// TwinCAT 3 PLC project Standard
// ProgramVersion: 3.1.4023.0
// libraries:
//   Tc2_MDP, * (Beckhoff Automation GmbH)
//   Tc2_Standard, * (Beckhoff Automation GmbH)
//   Tc2_SUPS, * (Beckhoff Automation GmbH)
//   Tc2_System, * (Beckhoff Automation GmbH)
//   Tc2_Utilities, * (Beckhoff Automation GmbH)
//   Tc3_BA2, * (Beckhoff Automation GmbH)
//   Tc3_BA2_Common, * (Beckhoff Automation GmbH)
//   Tc3_BACnetRev14, * (Beckhoff Automation GmbH)
//   Tc3_Module, * (Beckhoff Automation GmbH)
// project tree:
//   / PlcTask.TcTTO (not stored)
//   POUs/ MAIN.TcPOU (not stored)
//   Templates/DUTs/Enumerations/Building/ E_BA_BuildingMode.TcDUT
//   Templates/DUTs/Enumerations/Plant/AC/ E_BA_AC_OpMod01.TcDUT, E_BA_AC_OpMod02.TcDUT, E_BA_AC_SelSpErc.TcDUT
//   Templates/DUTs/Enumerations/Process/ E_BA_Process.TcDUT
//   Templates/DUTs/Enumerations/System/ E_BA_UPSType.TcDUT
//   Templates/DUTs/Enumerations/Universal/ E_BA_EnergyLvl.TcDUT, E_BA_EnergyLvlA.TcDUT, E_BA_EnergyLvlEx.TcDUT, E_BA_EnergyLvlExA.TcDUT, E_BA_MdltCmd.TcDUT, E_BA_OnOff.TcDUT, E_BA_OnOffA.TcDUT
//   Templates/DUTs/Types/Building/ ST_BA_BuildingAlarms.TcDUT
//   Templates/DUTs/Types/General/ ST_BA_GeneralSettings.TcDUT (not stored)
//   Templates/DUTs/Types/WeatherStation/ ST_BA_WeatherStation.TcDUT
//   Templates/GVLs/ BA2_Param.TcGVL
//   Templates/GVLs/DPAD/EventClasses/ EventClasses.TcGVL
//   Templates/GVLs/DPAD/Labels/1031/ LblAggregates1031.TcGVL, LblControl1031.TcGVL, LblFunctions1031.TcGVL
//   Templates/GVLs/DPAD/Labels/1033/ LblAggregates1033.TcGVL, LblControl1033.TcGVL, LblFunctions1033.TcGVL
//   Templates/GVLs/DPAD/Labels/Base/ LblAggregates.TcGVL (not stored), LblControl.TcGVL (not stored), LblFunctions.TcGVL (not stored)
//   Templates/GVLs/DPAD/Labels/Composition/ LblCmpAC.TcGVL, LblCmpGeneral.TcGVL, LblCmpHeating.TcGVL, LblCmpRoomAutomation.TcGVL, LblUniControl.TcGVL, LblUniFieldDevice.TcGVL
//   Templates/GVLs/DPAD/Texts/1031/ TxtEvent_1031.TcGVL, TxtPlant_1031.TcGVL, TxtTrade_1031.TcGVL
//   Templates/GVLs/DPAD/Texts/ TextPlants.TcGVL (not stored), Texts.TcGVL (not stored), TextTrades.TcGVL (not stored)
//   Templates/GVLs/Site/ Site.TcGVL (not stored)
//   Templates/POUs/Trade/AC/Aggregates/Cooler/Temperature/ FB_BA_AC_ColTSuACtrl.TcPOU, FB_BA_AC_ColT_02.TcPOU
//   Templates/POUs/Trade/AC/Aggregates/ERC/ FB_BA_AC_ErcTSuACtrl.TcPOU
//   Templates/POUs/Trade/AC/Aggregates/ERC/Plate/ FB_BA_AC_ErcPl_02.TcPOU
//   Templates/POUs/Trade/AC/Aggregates/PreHeater/ FB_BA_AC_PreHtr.TcPOU, FB_BA_AC_PreHtrTSuACtrl.TcPOU, FB_BA_AC_TRtCtrl.TcPOU
//   Templates/POUs/Trade/AC/ FB_BA_AC.TcPOU
//   Templates/POUs/Trade/AC/General/ FB_BA_AC_OpMod1St.TcPOU, FB_BA_AC_SumNgtCol.TcPOU
//   Templates/POUs/Trade/AC/Plants/ FB_BA_AHU_1St_PrHtr_ErcPl_Col.TcPOU
//   Templates/POUs/Trade/AC/Setpoint/Temperature/ FB_BA_AC_SpTRm_01.TcPOU, FB_BA_AC_TCasCtrl_01.TcPOU
//   Templates/POUs/Trade/General/Building/ FB_BA_BuildingAlarms.TcPOU, FB_BA_BuildingGlobal.TcPOU (not stored), FB_BA_BuildingMode.TcPOU
//   Templates/POUs/Trade/General/ControlCabinet/ FB_BA_ControlCabinet.TcPOU (not stored), FB_BA_ControlCabinetBasic.TcPOU (not stored)
//   Templates/POUs/Trade/General/EventClasses/ FB_BA_EvtGroups.TcPOU (not stored)
//   Templates/POUs/Trade/General/ FB_BA_General.TcPOU (not stored)
//   Templates/POUs/Trade/General/IFP/ FB_BA_IFP.TcPOU
//   Templates/POUs/Trade/General/IFP/Project/ FB_BA_ProjectEx.TcPOU (not stored)
//   Templates/POUs/Trade/General/Settings/ FB_BA_Settings.TcPOU, FB_BA_WeatherParamter.TcPOU (not stored)
//   Templates/POUs/Trade/HeatingSystem/Distribution/HeatingCircuit/ FB_BA_H_HtgCir01.TcPOU
//   Templates/POUs/Trade/HeatingSystem/ FB_BA_H.TcPOU
//   Templates/POUs/Trade/HeatingSystem/General/ FB_BA_HtgLmt.TcPOU, FB_BA_H_OpMod.TcPOU
//   Templates/POUs/Trade/HeatingSystem/Setpoint/ FB_BA_H_HtgCir_Sp.TcPOU
//   Templates/POUs/Trade/OutdoorDevices/ FB_BA_OD.TcPOU (not stored)
//   Templates/POUs/Universal/Aggregat/Analog/ FB_BA_ActuatorAnalog.TcPOU
//   Templates/POUs/Universal/Aggregat/Binary/ FB_BA_ActuatorCmd.TcPOU (not stored)
//   Templates/POUs/Universal/Control/AntiBlocking/ FB_BA_AntiBlocking.TcPOU
//   Templates/POUs/Universal/Control/EventClasses/ FB_BA_EvtCategory_SimpStand.TcPOU (not stored), FB_BA_EvtCategory_SimpStandExt.TcPOU (not stored)
//   Templates/POUs/Universal/Control/Hysteresis/ FB_BA_Hys_21.TcPOU
//   Templates/POUs/Universal/Control/Monitoring/ FB_BA_FdbAnalog.TcPOU, FB_BA_FdbBinary.TcPOU
//   Templates/POUs/Universal/Control/PID/ FB_BA_PID.TcPOU, FB_BA_PID_Sp.TcPOU
//   Templates/POUs/Universal/Control/Ramp/ FB_BA_RampLimitIncrease.TcPOU
//   Templates/POUs/Universal/Control/Scale/ FB_BA_Scale_02.TcPOU, FB_BA_Scale_04.TcPOU
//   Templates/POUs/Universal/Control/TimeDelay/ FB_BA_DlyOff.TcPOU, FB_BA_DlyOn.TcPOU
//   Templates/POUs/Universal/Control/Trend/ FB_BA_TrendLogging.TcPOU
//   Templates/POUs/Universal/Damper/2P/ FB_BA_Dmp2P.TcPOU
//   Templates/POUs/Universal/Motor/1st/ FB_BA_Mot1st.TcPOU
//   Templates/POUs/Universal/Motor/Control/ FB_BA_MotCtlExt.TcPOU
//   Templates/POUs/Universal/Pump/1st/ FB_BA_Pu1st.TcPOU
//   Templates/POUs/Universal/Sensor/ FB_BA_CombinationBI_BV.TcPOU (not stored), FB_BA_SensorAnalog_IO.TcPOU, FB_BA_SensorBinary_IO.TcPOU
//   Templates/POUs/Universal/Valve/ FB_BA_Vlv.TcPOU

// ---- Templates/DUTs/Enumerations/Building/E_BA_BuildingMode.TcDUT
{region '#Template'}
	{attribute 'Version' := '1.0.0.0'}
	{attribute 'Tags' := '"LCID": "1031", "Text": "DUT, Building, RA, OpMod, Mode"'}
	{attribute 'Tags' := '"LCID": "1033", "Text": "DUT, Building, RA, OpMod, Mode"'}
	{attribute 'Description' := '"LCID": "1031", "Text": "Gebäude-Betriebsart"'}
	{attribute 'Description' := '"LCID": "1033", "Text": "Building-operation-mode"'}
{endregion}

{attribute qualified_only}
TYPE E_BA_BuildingMode :
(
	eDefault		:= 1,
	eNightWatch		:= 2,
	eCleaning		:= 3
	
) UDINT;
END_TYPE

// ---- Templates/DUTs/Enumerations/Plant/AC/E_BA_AC_OpMod01.TcDUT
{region '#Template'}
	{attribute 'Version' := '1.0.0.0'}
	{attribute 'Tags' := '"LCID": "1031", "Text": "DUT, Plant, AC, OpMod"'}
	{attribute 'Tags' := '"LCID": "1033", "Text": "DUT, Plant, AC, OpMod"'}
	{attribute 'Description' := '"LCID": "1031", "Text": "Betriebsart Klimaanlage"'}
	{attribute 'Description' := '"LCID": "1033", "Text": "Operation Mode Air Conditioning"'}
{endregion}

{attribute qualified_only}
TYPE E_BA_AC_OpMod01 :
(
    Invalid							:= 0,
    eOff							:= 1,	// Aus							// Off
	eOn								:= 2,	// Ein							// On
    eEmergency						:= 3,	// Notfall						// Emergency
    eFrost							:= 4,	// Frost						// Frost
    eSmokeExtractionProgramm		:= 5,	// Entrauchung Programm			// Smoke extraction programm
    eSmokeExtractionSupplyAir		:= 6,	// Entrauchung Zuluft			// Smoke extraction supply air
    eSmokeExtractionExhaustAir		:= 7,	// Entrauchung Fortluft			// Smoke extraction exhaust air
    eFire							:= 8,	// Feuer						// Fire
    eNightCooling					:= 9,	// Nachtkühlung					// Night cooling
    eCoolDownProtection				:= 10,	// Stützbetrieb,Auskühlschutz	// Cool down protection
    eOverHeatingProtection			:= 11,	// Überhitzungsschutz			// Over heating protection
    eAlarm							:= 12,	// Störung						// Alarm
    eForcedVentilation				:= 13,	// Zwangsbelüftung				// Forced ventilation
    eCentralSwitchOff				:= 14	// Zentralabschaltung			// Central switch-off
) UDINT;
END_TYPE

// ---- Templates/DUTs/Enumerations/Plant/AC/E_BA_AC_OpMod02.TcDUT
{region '#Template'}
	{attribute 'Version' := '1.0.0.0'}
	{attribute 'Tags' := '"LCID": "1031", "Text": "DUT, Plant, AC, OpMod"'}
	{attribute 'Tags' := '"LCID": "1033", "Text": "DUT, Plant, AC, OpMod"'}
	{attribute 'Description' := '"LCID": "1031", "Text": "Betriebsart Klimaanlage"'}
	{attribute 'Description' := '"LCID": "1033", "Text": "Operation Mode Air Conditioning"'}
{endregion}

{attribute qualified_only}
TYPE E_BA_AC_OpMod02 :
(
    Invalid							:= 0,
    eOff							:= 1,	// Aus//Off
    eStep1							:= 2,	// Stufe 1						// Step 1
    eStep2							:= 3,	// Stufe 2						// Step 2
    eStep3							:= 4,	// Stufe 3						// Step 3
    eEmergency						:= 5,	// Notfall						// Emergency
    eFrost							:= 6,	// Frost						// Frost
    eSmokeExtractionProgramm		:= 7,	// Entrauchung Programm			// Smoke extraction program
    eSmokeExtractionSupplyAir		:= 8,	// Entrauchung Zuluft			// Smoke extraction supply air
    eSmokeExtractionExhaustAir		:= 9,	// Entrauchung Fortluft			// Smoke extraction exhaust air
    eFire							:= 10,	// Feuer						// Fire
    eNightCooling					:= 11,	// Nachtkühlung					// Night cooling
    eCoolDownProtection				:= 12,	// Stützbetrieb,Auskühlschutz	// Cool down protection
    eOverHeatingProtection			:= 13,	// Überhitzungsschutz			// Over heating protection
    eAlarm							:= 14,	// Störung						// Alarm
    eForcedVentilation				:= 15,	// Zwangsbelüftung				// Forced ventilation
    eCentralSwitchOff				:= 16	// Zentralabschaltung			// Central switch-off
) UDINT;
END_TYPE

// ---- Templates/DUTs/Enumerations/Plant/AC/E_BA_AC_SelSpErc.TcDUT
{region '#Template'}
	{attribute 'Version' := '1.0.0.0'}
	{attribute 'Tags' := '"LCID": "1031", "Text": "DUT, Plant, AC, Setpoint"'}
	{attribute 'Tags' := '"LCID": "1033", "Text": "DUT, Plant, AC, Setpoint"'}
	{attribute 'Description' := '"LCID": "1031", "Text": "Auswahl Sollwert Energie Rückgewinnung"'}
	{attribute 'Description' := '"LCID": "1033", "Text": "Selection setpoint energy recovery"'}
{endregion}

{attribute 'qualified_only'}
TYPE E_BA_AC_SelSpErc :
(
	eAction				:= 1,	//	E_BA_Action.eDirect = SpCol, E_BA_Action.eReverse = SpHtg, 
	eAverageHtgCol		:= 2	
) UDINT;
END_TYPE

// ---- Templates/DUTs/Enumerations/Process/E_BA_Process.TcDUT
{region '#Template'}
	{attribute 'Version' := '1.0.0.0'}
	{attribute 'Tags' := '"LCID": "1031", "Text": "DUT, Process, AC, Steps"'}
	{attribute 'Tags' := '"LCID": "1033", "Text": "DUT, Process, AC, Steps"'}
	{attribute 'Description' := '"LCID": "1031", "Text": "AC Status"'}
	{attribute 'Description' := '"LCID": "1033", "Text": "AC states"'}
{endregion}

{attribute 'qualified_only'}
TYPE E_BA_Process :
(
	Invalid							:= 0,
	eOff							:= 1,	
	ePreRinse						:= 2,
	eDriveDamper					:= 3,
	eFanSupplyAir					:= 4,
	eFanExtractAir					:= 5,
	eEnablingTemperatureControl		:= 6,
	eEnablingHumidityControl		:= 7,
	eEnablingLimitMonitoring		:= 8
) UDINT;
END_TYPE

// ---- Templates/DUTs/Enumerations/System/E_BA_UPSType.TcDUT
{region '#Template'}
	{attribute 'Version' := '0.0.1.0'}
	{attribute 'Tags' := '"LCID": "1031", "Text": "DUT, System, UPS"'}
	{attribute 'Tags' := '"LCID": "1033", "Text": "DUT, System, UPS"'}
	{attribute 'Description' := '"LCID": "1031", "Text": "Einstellung USV"'}
	{attribute 'Description' := '"LCID": "1033", "Text": "Settings UPS"'}
{endregion}

{attribute 'qualified_only'}
{attribute 'strict'}
TYPE E_BA_UPSType :
(
	eNone := 0,
	
	eCX50x0,
	eCX51x0,
	eCX81xx,
	eCX9020_U900,
	eCB3011
);
END_TYPE

// ---- Templates/DUTs/Enumerations/Universal/E_BA_EnergyLvl.TcDUT
{region '#Template'}
	{attribute 'Version' := '1.0.0.0'}
	{attribute 'Tags' := '"LCID": "1031", "Text": "DUT, Room automation, Heating system"'}
	{attribute 'Tags' := '"LCID": "1033", "Text": "DUT, Room automation, Heating system"'}
	{attribute 'Description' := '"LCID": "1031", "Text": "Betriebsart Energieniveau"'}
	{attribute 'Description' := '"LCID": "1033", "Text": "Operating mode Energy level"'}
{endregion}

{attribute qualified_only}
TYPE E_BA_EnergyLvl :
(
	eProtection		:= 1,
	eEconomy		:= 2,
	eComfort		:= 3
	
) UDINT;
END_TYPE

// ---- Templates/DUTs/Enumerations/Universal/E_BA_EnergyLvlA.TcDUT
{region '#Template'}
	{attribute 'Version' := '1.0.0.0'}
	{attribute 'Tags' := '"LCID": "1031", "Text": "DUT, Room automation, Heating system"'}
	{attribute 'Tags' := '"LCID": "1033", "Text": "DUT, Room automation, Heating system"'}
	{attribute 'Description' := '"LCID": "1031", "Text": "Betriebsart Energieniveau"'}
	{attribute 'Description' := '"LCID": "1033", "Text": "Operating mode Energy level"'}
{endregion}

{attribute qualified_only}
TYPE E_BA_EnergyLvlA :
(
	eAutomatic		:= 1,
	eProtection		:= 2,
	eEconomy		:= 3,
	eComfort		:= 4
	
) UDINT;
END_TYPE

// ---- Templates/DUTs/Enumerations/Universal/E_BA_EnergyLvlEx.TcDUT
{region '#Template'}
	{attribute 'Version' := '1.0.0.0'}
	{attribute 'Tags' := '"LCID": "1031", "Text": "DUT, Room automation, Heating system"'}
	{attribute 'Tags' := '"LCID": "1033", "Text": "DUT, Room automation, Heating system"'}
	{attribute 'Description' := '"LCID": "1031", "Text": "Betriebsart Energieniveau"'}
	{attribute 'Description' := '"LCID": "1033", "Text": "Operating mode Energy level"'}
{endregion}

{attribute qualified_only}
TYPE E_BA_EnergyLvlEx :
(
	eProtection			:= 1,
	eEconomy			:= 2,
	ePreComfort			:= 3,
	eComfort			:= 4
	
) UDINT;
END_TYPE

// ---- Templates/DUTs/Enumerations/Universal/E_BA_EnergyLvlExA.TcDUT
{region '#Template'}
	{attribute 'Version' := '1.0.0.0'}
	{attribute 'Tags' := '"LCID": "1031", "Text": "DUT, Room automation, Heating system"'}
	{attribute 'Tags' := '"LCID": "1033", "Text": "DUT, Room automation, Heating system"'}
	{attribute 'Description' := '"LCID": "1031", "Text": "Betriebsart Energieniveau"'}
	{attribute 'Description' := '"LCID": "1033", "Text": "Operating mode Energy level"'}
{endregion}

{attribute qualified_only}
TYPE E_BA_EnergyLvlExA :
(
	eAutomatic		:= 1,
	eProtection		:= 2,
	eEconomy		:= 3,
	ePreComfort		:= 4,
	eComfort		:= 5
	
) UDINT;
END_TYPE

// ---- Templates/DUTs/Enumerations/Universal/E_BA_MdltCmd.TcDUT
{region '#Template'}
	{attribute 'Version' := '1.0.0.0'}
	{attribute 'Tags' := '"LCID": "1031", "Text": "DUT, Operation mode, Universal, Modulation"'}
	{attribute 'Tags' := '"LCID": "1033", "Text": "DUT, Operation mode, Universal, Modulation"'}
	{attribute 'Description' := '"LCID": "1031", "Text": "Modulationsbefehle"'}
	{attribute 'Description' := '"LCID": "1033", "Text": "modulation commands"'}
{endregion}

{attribute 'qualified_only'}
TYPE E_BA_MdltCmd :
(
	eOff			:= 1,
	eOn				:= 2,
	eMin			:= 3,
	eMax			:= 4
	
) UDINT;
END_TYPE

// ---- Templates/DUTs/Enumerations/Universal/E_BA_OnOff.TcDUT
{region '#Template'}
	{attribute 'Version' := '1.0.0.0'}
	{attribute 'Tags' := '"LCID": "1031", "Text": "DUT, Operation mode, Universal, On, Off"'}
	{attribute 'Tags' := '"LCID": "1033", "Text": "DUT, Operation mode, Universal, On, Off"'}
	{attribute 'Description' := '"LCID": "1031", "Text": "Betriebsart Ein Aus"'}
	{attribute 'Description' := '"LCID": "1033", "Text": "Operating on off"'}
{endregion}

{attribute qualified_only}
TYPE E_BA_OnOff :
(
	eOff			:= 1,
	eOn				:= 2
	
) UDINT;
END_TYPE

// ---- Templates/DUTs/Enumerations/Universal/E_BA_OnOffA.TcDUT
{region '#Template'}
	{attribute 'Version' := '1.0.0.0'}
	{attribute 'Tags' := '"LCID": "1031", "Text": "DUT, Operation mode, Universal, On, Off"'}
	{attribute 'Tags' := '"LCID": "1033", "Text": "DUT, Operation mode, Universal, On, Off"'}
	{attribute 'Description' := '"LCID": "1031", "Text": "Betriebsart Ein Aus Auto"'}
	{attribute 'Description' := '"LCID": "1033", "Text": "Operating on off auto"'}
{endregion}

{attribute qualified_only}
TYPE E_BA_OnOffA :
(
	eAutomatic		:= 1,
	eOff			:= 2,
	eOn				:= 3
	
) UDINT;
END_TYPE

// ---- Templates/DUTs/Types/Building/ST_BA_BuildingAlarms.TcDUT
{region '#Template'}
	{attribute 'Version' := '0.0.1.0'}
	{attribute 'Tags' := '"LCID": "1031", "Text": "Types, Publisher, Subscriber, Building, General, Alarms, Events"'}
	{attribute 'Tags' := '"LCID": "1033", "Text": "Types, Publisher, Subscriber, Building, General, Alarms, Events"'}
	{attribute 'Description' := '"LCID": "1031", "Text": "Gebäude-Alarme und -Events"'}
	{attribute 'Description' := '"LCID": "1033", "Text": "Building-alarms and -events"'}
{endregion}
TYPE ST_BA_BuildingAlarms :
STRUCT
	bBurglary				: BOOL;
	bFireAlert				: BOOL;
	bCentralOff				: BOOL;
	bForcedVentilation		: BOOL;
	bSmokeExtraction		: BOOL;
END_STRUCT
END_TYPE

// ---- Templates/DUTs/Types/WeatherStation/ST_BA_WeatherStation.TcDUT
{region '#Template'}
	{attribute 'Version' := '0.0.1.0'}
	{attribute 'Tags' := '"LCID": "1031", "Text": "Types, Publisher, Subscriber, Weather, Data"'}
	{attribute 'Tags' := '"LCID": "1033", "Text": "Types, Publisher, Subscriber, Weather, Data"'}
	{attribute 'Description' := '"LCID": "1031", "Text": "Daten Wetterstation"'}
	{attribute 'Description' := '"LCID": "1033", "Text": "Weatherstation-data"'}
{endregion}
TYPE ST_BA_WeatherStation :
STRUCT
	bDisturb				: BOOL;
	fLatitude				: REAL;				// [°]
	fLongitude				: REAL;				// [°]
	fSunAzimuth				: REAL;				// [°]
	fSunElevation			: REAL;				// [°]
	bRain					: BOOL;
	stDateTime				: TIMESTRUCT;
	fOutsideTemperature		: REAL;				// [°C]
	fDewPointTemperature	: REAL;				// [°C]		 
	fPressureAbs			: REAL;				// [hPa]
	fPressureRel			: REAL;				// [hPa]			 
	fHumidityAbs			: REAL;				// [%rF]
	fHumidityRel			: REAL;				// [g/m³]			 
	fBrightnessEast			: REAL;				// [Lux]
	fBrightnessNorth		: REAL;				// [Lux]
	fBrightnessSouth		: REAL;				// [Lux]
	fBrightnessWest			: REAL;				// [Lux]			 
	fDawn					: REAL;				// [Lux] 
	fGlobalRadiation		: REAL;				// [W/m²]			 
	fWindDirection			: REAL;				// [°]
	fWindSpeed				: REAL;				// [m/s]
END_STRUCT
END_TYPE

// ---- Templates/GVLs/BA2_Param.TcGVL
{region '#Template'}
	{attribute 'Version' := '1.0.0.0'}
	{attribute 'Tags' := '"LCID": "1031", "Text": "GVL, Constants"'}
	{attribute 'Tags' := '"LCID": "1033", "Text": "GVL, Constants"'}
	{attribute 'Description' := '"LCID": "1031", "Text": "Globale Konstanten"'}
	{attribute 'Description' := '"LCID": "1033", "Text": "Global constants"'}
{endregion}

{attribute 'qualified_only'}
{attribute 'strict'}
VAR_GLOBAL CONSTANT 
	fAP                					: REAL 						:= 1013.25;	// Hydrostatischer Luftdruck	//	atmospheric pressure

	nDefTimeDelay_ToAbnormal			: UDINT						:= 1;
	nDefTimeDelay_ToNormal				: UDINT						:= 0;

	fDefCOVIncrement					: REAL						:= 0.1;	

	fDefLimitDeadband					: REAL						:= 0.0;

	nLoop_DefOpMode						: E_BA_PIDMode				:= E_BA_PIDMode.eP1ID;	
	
	{warning disable C0228}
	stTrend_DefStartTime				: ST_BA_DateTime			;(*:= F_BA_ToSTDateTime(DT#2099-01-01-00:13);*)
	stTrend_DefStopTime					: ST_BA_DateTime			;(* := F_BA_ToSTDateTime(DT#2099-01-01-00:13);*)
	{warning restore C0228}
	nTrend_BufferSize					: UDINT						:= 500;	// Count of entries in a Trend-Buffer	
	bTrend_DefLogEnable					: BOOL						:= FALSE;
	bTrend_DefStopOnFull				: BOOL						:= FALSE;
	nTrend_DefLogInterval				: UDINT						:= 90;	// (in [s])
	nTrend_DefNotificationThreshold		: UDINT						:= 50;
	eTrend_DefLoggingType				: E_BA_LoggingType			:= E_BA_LoggingType.ePolled;				
END_VAR

// ---- Templates/GVLs/DPAD/EventClasses/EventClasses.TcGVL
{region '#Template'}
	{attribute 'Version' := '1.0.0.0'}
	{attribute 'Tags' := '"LCID": "1031", "Text": "General, Notification classes, Event classes"'}
	{attribute 'Tags' := '"LCID": "1033", "Text": "General, Notification classes, Event classes"'}
	{attribute 'Description' := '"LCID": "1031", "Text": "Ereignisklassen"'}
	{attribute 'Description' := '"LCID": "1033", "Text": "Event classes"'}
{endregion}

{attribute 'qualified_only'}
VAR_GLOBAL CONSTANT
	LifeSafetySimple				: UDINT	:= 12;
	LifeSafetyStandard				: UDINT	:= 11;
	LifeSafetyExtended				: UDINT	:= 10;
                            		
	AlarmTechnicalSimple			: UDINT	:= 22;
	AlarmTechnicalStandard			: UDINT	:= 21;
	AlarmTechnicalExtended			: UDINT	:= 20;	
	
	DisturbanceSimple				: UDINT	:= 52;
	DisturbanceStandard				: UDINT	:= 51;
	DisturbanceExtended				: UDINT	:= 50;
		
	MaintenanceSimple				: UDINT	:= 92;
	MaintenanceStandard				: UDINT	:= 91;
	MaintenanceExtended				: UDINT	:= 90;
	
	NotificationSimple				: UDINT	:= 132;
	NotificationStandard			: UDINT	:= 131;
	
	OtherSimple						: UDINT	:= 182;
	OtherStandard					: UDINT	:= 181;
END_VAR

// ---- Templates/GVLs/DPAD/Labels/1031/LblAggregates1031.TcGVL
{region '#Template'}
	{attribute 'Version' := '1.0.0.0'}
	{attribute 'Tags' := '"LCID": "1031", "Text": "GVL, AKS, Labels, ObjectName, Description"'}
	{attribute 'Tags' := '"LCID": "1033", "Text": "GVL, DPAD, Labels, ObjectName, Description"'}
	{attribute 'Description' := '"LCID": "1031", "Text": "Anlagenkennzeichnungssystem, Labels Aggregate"'}
	{attribute 'Description' := '"LCID": "1033", "Text": "Data Point Addressing Description, Labels aggregate"'}
{endregion}

{attribute 'global_init_slot' := '40510'}
VAR_GLOBAL
  LblAggregates_FunctionallyIndependentEequipment                 :FB_BA_Label:=( sObjName:='FEE', sDescr:='Funktional eigenständige Einrichtung');
  LblAggregates_SelfContainedControlUnit                          :FB_BA_Label:=( sObjName:='ASR', sDescr:='Autarke Steuer- oder Regeleinheit');
  LblAggregates_ControlCabinet                                    :FB_BA_Label:=( sObjName:='SSK', sDescr:='Schaltschrank (gewerkespezifisch)');
//330 Türen, Tore, Fenster, Sonnenschutz
  LblAggregates_WindowDrive                                       :FB_BA_Label:=( sObjName:='FEN', sDescr:='Fenster (Antrieb)');
  LblAggregates_WindowContact                                     :FB_BA_Label:=( sObjName:='FEK', sDescr:='Fensterkontakt');
  LblAggregates_Blind                                             :FB_BA_Label:=( sObjName:='JAL', sDescr:='Jalousie');
  LblAggregates_Awning                                            :FB_BA_Label:=( sObjName:='MAR', sDescr:='Markise');
  LblAggregates_RollerShutters                                    :FB_BA_Label:=( sObjName:='ROL', sDescr:='Rollläden');
  LblAggregates_Gate                                              :FB_BA_Label:=( sObjName:='TOR', sDescr:='Tor');
  LblAggregates_Door                                              :FB_BA_Label:=( sObjName:='TÜR', sDescr:='Tür');
  LblAggregates_DoorContact                                       :FB_BA_Label:=( sObjName:='TÜK', sDescr:='Türkontakt');
  LblAggregates_Blackout                                          :FB_BA_Label:=( sObjName:='VER', sDescr:='Verdunklung');
//412 Wasseranlagen
  LblAggregates_TraceHeating                                      :FB_BA_Label:=( sObjName:='BGH', sDescr:='Begleitheizung');
  LblAggregates_ElectricHeating                                   :FB_BA_Label:=( sObjName:='EWH', sDescr:='Elektroheizung (TWW–Bereitung)');
  LblAggregates_WaterFilter                                       :FB_BA_Label:=( sObjName:='WFL', sDescr:='Wasserfilter');
//421 Wärmeerzeugungsanlagen
  LblAggregates_Furnace                                           :FB_BA_Label:=( sObjName:='HZK', sDescr:='Heizkessel');
  LblAggregates_HeatExchanger                                     :FB_BA_Label:=( sObjName:='WÜT', sDescr:='Wärmeübertrager');
//430 Lufttechnische Anlagen und Kälteanlagen
  LblAggregates_FanExhaustAir                                     :FB_BA_Label:=( sObjName:='FOV', sDescr:='Fortluftventilator');
  LblAggregates_Airwasher                                         :FB_BA_Label:=( sObjName:='LWS', sDescr:='Luftwäscher');
  LblAggregates_Humidifier                                        :FB_BA_Label:=( sObjName:='BEF', sDescr:='Befeuchter');
  LblAggregates_HumidifierPump                                    :FB_BA_Label:=( sObjName:='BFP', sDescr:='Befeuchterpumpe');
  LblAggregates_FireDamper                                        :FB_BA_Label:=( sObjName:='BSK', sDescr:='Brandschutzklappe, -ventil');
  LblAggregates_SmokeProtectionDamper                             :FB_BA_Label:=( sObjName:='RSK', sDescr:='Rauchschutzklappe');
  LblAggregates_SmokeExtractorDamper                              :FB_BA_Label:=( sObjName:='ERK', sDescr:='Entrauchungsklappe');
  LblAggregates_CeilingSwirlDiffuser                              :FB_BA_Label:=( sObjName:='DDA', sDescr:='Deckendrallauslass');
  LblAggregates_RoofAirHeater                                     :FB_BA_Label:=( sObjName:='DLA', sDescr:='Deckenlufterhitzer');
  LblAggregates_DirectEvaporator                                  :FB_BA_Label:=( sObjName:='DVD', sDescr:='Direktverdampfer');
  LblAggregates_ElectricalAirHeater                               :FB_BA_Label:=( sObjName:='ELH', sDescr:='Elektrolufterhitzer');
  LblAggregates_ElectricReHeater                                  :FB_BA_Label:=( sObjName:='ENH', sDescr:='Elektronacherhitzer');
  LblAggregates_ElectricaPreHeater                                :FB_BA_Label:=( sObjName:='EVH', sDescr:='Elektrovorerhitzer');
  LblAggregates_HeaterGeneral                                     :FB_BA_Label:=( sObjName:='ERH', sDescr:='Erhitzer');
  LblAggregates_FanExtractAir                                     :FB_BA_Label:=( sObjName:='ABV', sDescr:='Abluftventilator');
  LblAggregates_InductionDevice                                   :FB_BA_Label:=( sObjName:='IND', sDescr:='Induktionsgerät');
  LblAggregates_RefrigerantDryer                                  :FB_BA_Label:=( sObjName:='KTR', sDescr:='Kältetrockner');
  LblAggregates_CirculatorySystem                                 :FB_BA_Label:=( sObjName:='KVS', sDescr:='KVS (WRG über Kreislaufverbundsysteme)');
  LblAggregates_AirFilterOutsideAir                               :FB_BA_Label:=( sObjName:='LFI', sDescr:='Außenluftfilter');
  LblAggregates_AirFilterSupplyAir                                :FB_BA_Label:=( sObjName:='LFI', sDescr:='Zuluftfilter');
  LblAggregates_AirFilterExhaustAir                               :FB_BA_Label:=( sObjName:='LFI', sDescr:='Fortluftfilter');
  LblAggregates_AirFilterExtractAir                               :FB_BA_Label:=( sObjName:='LFI', sDescr:='Abluftfilter');
  LblAggregates_AirFilter                                         :FB_BA_Label:=( sObjName:='LFI', sDescr:='Luftfilter');
  LblAggregates_VentilationDamper                                 :FB_BA_Label:=( sObjName:='LKL', sDescr:='Lüftungsklappe');
  LblAggregates_VentilationDamperOutsideAir                       :FB_BA_Label:=( sObjName:='LKL', sDescr:='Außenluftklappe');
  LblAggregates_VentilationDamperExhaustAir                       :FB_BA_Label:=( sObjName:='LKL', sDescr:='Fortluftklappe');
  LblAggregates_VentilationDamperMixAir                           :FB_BA_Label:=( sObjName:='LKL', sDescr:='Mischluftklappe');
  LblAggregates_VentilationDamperSupplyAir                        :FB_BA_Label:=( sObjName:='LKL', sDescr:='Zuluftklappe');
  LblAggregates_VentilationDamperBypassAir                        :FB_BA_Label:=( sObjName:='LKL', sDescr:='Bypassklappe');
  LblAggregates_Pump                                              :FB_BA_Label:=( sObjName:='PPE', sDescr:='Pumpe');
  LblAggregates_RecirculatingAirCoolingDevice                     :FB_BA_Label:=( sObjName:='ULK', sDescr:='Umluftkühlgerät');
  LblAggregates_FanRecirculatingAir                               :FB_BA_Label:=( sObjName:='UMV', sDescr:='Umluftventilator');
  LblAggregates_UvFilter                                          :FB_BA_Label:=( sObjName:='UVF', sDescr:='UV-Filter');
  LblAggregates_VariableFlowRateController                        :FB_BA_Label:=( sObjName:='VVR', sDescr:='Variabler Volumenstromregler');
  LblAggregates_WaterAirHeater                                    :FB_BA_Label:=( sObjName:='WLH', sDescr:='Wasserlufterhitzer');
  LblAggregates_WaterReHeater                                     :FB_BA_Label:=( sObjName:='WNH', sDescr:='Wassernacherhitzer');
  LblAggregates_WaterPreHeater                                    :FB_BA_Label:=( sObjName:='WVH', sDescr:='Wasservorerhitzer');
  LblAggregates_HeatRecovery                                      :FB_BA_Label:=( sObjName:='WRG', sDescr:='Wärmerückgewinnung');
  LblAggregates_FanSupplyAir                                      :FB_BA_Label:=( sObjName:='ZUV', sDescr:='Zuluftventilator');
  LblAggregates_SmokeExtractionSystems                            :FB_BA_Label:=( sObjName:='ERA', sDescr:='Entrauchungsanlagen');
  LblAggregates_SmokeExtractionVentilator                         :FB_BA_Label:=( sObjName:='ERV', sDescr:='Entrauchungsventilator');
  LblAggregates_VentWindow                                        :FB_BA_Label:=( sObjName:='NSF', sDescr:='Nachströmfenster');
  LblAggregates_VentFlap                                          :FB_BA_Label:=( sObjName:='NSK', sDescr:='Nachströmklappe');
  LblAggregates_VentDoor                                          :FB_BA_Label:=( sObjName:='NST', sDescr:='Nachströmtür');
  LblAggregates_WakeFan                                           :FB_BA_Label:=( sObjName:='NSV', sDescr:='Nachströmventilator');
//434 Kälteanlagen
  LblAggregates_GlycoOilProtector                                 :FB_BA_Label:=( sObjName:='GLP', sDescr:='Glykol/Ölprotektor');
  LblAggregates_Chiller                                           :FB_BA_Label:=( sObjName:='KMA', sDescr:='Kältemaschine');
  LblAggregates_ReCoolingPlant                                    :FB_BA_Label:=( sObjName:='RKW', sDescr:='Rückkühlwerk');
//440 Starkstromanlagen
  LblAggregates_GeneralPowerSupply                                :FB_BA_Label:=( sObjName:='ASV', sDescr:='Allgemeine Spannungsversorgung');
  LblAggregates_CombindeHeatPowerStation                          :FB_BA_Label:=( sObjName:='BHK', sDescr:='Blockheizkraftwerk');
  LblAggregates_CompensationSystem                                :FB_BA_Label:=( sObjName:='KOA', sDescr:='Kompensationsanlage');
  LblAggregates_CouplingSwitch                                    :FB_BA_Label:=( sObjName:='KUS', sDescr:='Kuppelschalter');
  LblAggregates_LoadBreakSwitch                                   :FB_BA_Label:=( sObjName:='LTS', sDescr:='Lasttrennschalter');
  LblAggregates_CircuitBreaker                                    :FB_BA_Label:=( sObjName:='LSS', sDescr:='Leistungsschalter');
  LblAggregates_NetworkAnalyser                                   :FB_BA_Label:=( sObjName:='NAG', sDescr:='Netzanalysegerät');
  LblAggregates_EmergencyPoweGeneratorUnit                        :FB_BA_Label:=( sObjName:='NSG', sDescr:='Notstromaggregat');
  LblAggregates_EmergencyLighting                                 :FB_BA_Label:=( sObjName:='SIB', sDescr:='Sicherheitsbeleuchtung');
  LblAggregates_SafetyPowerSupply                                 :FB_BA_Label:=( sObjName:='SSV', sDescr:='Sicherheitsspannungsversorgung');
  LblAggregates_Transformer                                       :FB_BA_Label:=( sObjName:='TRF', sDescr:='Transformator');
  LblAggregates_UninterruptiblePowerSupply                        :FB_BA_Label:=( sObjName:='USV', sDescr:='Unterbrechungsfreie Spannungsversorgung');
//450 Fernmelde- und informationstechnische Anlagen
  LblAggregates_CentralFireAlarmSystem                            :FB_BA_Label:=( sObjName:='BMZ', sDescr:='Brandmeldezentrale');
  LblAggregates_FireControlPanel                                  :FB_BA_Label:=( sObjName:='FWT', sDescr:='Feuerwehrtableau');
  LblAggregates_KitchenTableau                                    :FB_BA_Label:=( sObjName:='KÜT', sDescr:='Küchentableau');
  LblAggregates_SmokeDetector                                     :FB_BA_Label:=( sObjName:='RME', sDescr:='Rauchmelder');
  LblAggregates_SmokeProtectionScreen                             :FB_BA_Label:=( sObjName:='RSV', sDescr:='Rauchschutzvorhang');
  LblAggregates_VoiceAlarmCentre                                  :FB_BA_Label:=( sObjName:='SAZ', sDescr:='Sprachalarmierungszentrale');
  LblAggregates_Tableau                                           :FB_BA_Label:=( sObjName:='TBL', sDescr:='Tableau (allgemein)');
//460 Förderanlagen
  LblAggregates_LiftGeneral                                       :FB_BA_Label:=( sObjName:='AZA', sDescr:='Aufzug allgemein');
  LblAggregates_GoodsLift                                         :FB_BA_Label:=( sObjName:='AZL', sDescr:='Lastenaufzug');
  LblAggregates_PassengerLift                                     :FB_BA_Label:=( sObjName:='AZP', sDescr:='Personenaufzug');
//470 Nutzerspezifische Anlagen
  LblAggregates_FumeCupboard                                      :FB_BA_Label:=( sObjName:='DIG', sDescr:='Digestorium');
  LblAggregates_Compressor                                        :FB_BA_Label:=( sObjName:='KOM', sDescr:='Kompressor');
  LblAggregates_ProgrammableLogicControllers                      :FB_BA_Label:=( sObjName:='SPS', sDescr:='Speicherprogrammierbare Steuerung');
//479 Nutzerspezifische Anlage, Wetterstation
  LblAggregates_RainSensor                                        :FB_BA_Label:=( sObjName:='RGM', sDescr:='Regenmelder');
  LblAggregates_SolarRadiation                                    :FB_BA_Label:=( sObjName:='SES', sDescr:='Sonneneinstrahlung');
  LblAggregates_WeatherStation                                    :FB_BA_Label:=( sObjName:='WST', sDescr:='Wetterstation');
  LblAggregates_WindSpeed                                         :FB_BA_Label:=( sObjName:='WDG', sDescr:='Windgeschwindigkeit');
  LblAggregates_WindDirection                                     :FB_BA_Label:=( sObjName:='WDR', sDescr:='Windrichtung');
  LblAggregates_WindForce                                         :FB_BA_Label:=( sObjName:='WDS', sDescr:='Windstärke');
  LblAggregates_Brightness                                        :FB_BA_Label:=( sObjName:='HEL', sDescr:='Helligkeit');
  LblAggregates_Dawn                                              :FB_BA_Label:=( sObjName:='HED', sDescr:='Dämmerungshelligkeit');
  LblAggregates_PressureAbsolute                                  :FB_BA_Label:=( sObjName:='LUA', sDescr:='Luftdruck absolut');
  LblAggregates_PressureRelative                                  :FB_BA_Label:=( sObjName:='LUR', sDescr:='Luftdruck relativ');
  LblAggregates_GeoLatitude                                       :FB_BA_Label:=( sObjName:='BRG', sDescr:='Breitengrad');
  LblAggregates_GeoLongitude                                      :FB_BA_Label:=( sObjName:='LAG', sDescr:='Längengrad');
  LblAggregates_SunAzimuth                                        :FB_BA_Label:=( sObjName:='SST', sDescr:='Sonnenstand');
  LblAggregates_SunElevation                                      :FB_BA_Label:=( sObjName:='SEL', sDescr:='Elevation');
//480 Gebäudeautomation
  LblAggregates_SystemSwitch                                      :FB_BA_Label:=( sObjName:='ANL', sDescr:='Anlagenschalter');
  LblAggregates_AutomationStationEquipment                        :FB_BA_Label:=( sObjName:='ASE', sDescr:='Automationsstationseinrichtung');
  LblAggregates_BusLineCoupler                                    :FB_BA_Label:=( sObjName:='BUS', sDescr:='Bus-Linien-Koppler');
  LblAggregates_DataInterfaceUnit                                 :FB_BA_Label:=( sObjName:='DSE', sDescr:='Datenschnittstelleneinheit');
  LblAggregates_FieldbusModule                                    :FB_BA_Label:=( sObjName:='FBM', sDescr:='Feldbusmodul');
  LblAggregates_InformationFocalPoint                             :FB_BA_Label:=( sObjName:='ISP', sDescr:='Informationsschwerpunkt');
  LblAggregates_ManagementAndControlEquipment                     :FB_BA_Label:=( sObjName:='MBE', sDescr:='Management- und Bedieneinrichtung');
//481 GA-Sensorik – Temperatur
  LblAggregates_TemperatureGasEmission                            :FB_BA_Label:=( sObjName:='TAG', sDescr:='Abgastemperatur');
  LblAggregates_TemperatureExtractAir                             :FB_BA_Label:=( sObjName:='TAB', sDescr:='Ablufttemperatur');
  LblAggregates_TemperatureOutside                                :FB_BA_Label:=( sObjName:='TAU', sDescr:='Außentemperatur');
  LblAggregates_TemperatureExhaustAir                             :FB_BA_Label:=( sObjName:='TFO', sDescr:='Fortlufttemperatur');
  LblAggregates_FrostProtectionMonitor                            :FB_BA_Label:=( sObjName:='FSW', sDescr:='Frostschutzwächter');
  LblAggregates_TemperatureMixedAir                               :FB_BA_Label:=( sObjName:='TMI', sDescr:='Mischlufttemperatur');
  LblAggregates_TemperatureRoomAir                                :FB_BA_Label:=( sObjName:='TRU', sDescr:='Raumtemperatur');
  LblAggregates_TemperatureReturnFlow                             :FB_BA_Label:=( sObjName:='TRL', sDescr:='Rücklauftemperatur');
  LblAggregates_LimiterSafetyTemperature                          :FB_BA_Label:=( sObjName:='STB', sDescr:='Sicherheitstemperaturbegrenzer');
  LblAggregates_MonitorSafetyTemperature                          :FB_BA_Label:=( sObjName:='STW', sDescr:='Sicherheitstemperaturwächter');
  LblAggregates_TemperatureStorage                                :FB_BA_Label:=( sObjName:='TSP', sDescr:='Speichertemperatur');
  LblAggregates_TemperatureDewPoint                               :FB_BA_Label:=( sObjName:='TTP', sDescr:='Taupunkttemperatur');
  LblAggregates_MonitorDewPoint                                   :FB_BA_Label:=( sObjName:='TPW', sDescr:='Taupunktwächter');
  LblAggregates_TemperatureAfterCooler                            :FB_BA_Label:=( sObjName:='TNK', sDescr:='Temperatur nach Kühler');
  LblAggregates_TemperatureAfterPreHeater                         :FB_BA_Label:=( sObjName:='TNV', sDescr:='Temperatur nach Vorerhitzer');
  LblAggregates_TemperatureAfterHeatRecovery                      :FB_BA_Label:=( sObjName:='TNW', sDescr:='Temperatur nach Wärmerückgewinnung');
  LblAggregates_Thermostat                                        :FB_BA_Label:=( sObjName:='THM', sDescr:='Thermostat');
  LblAggregates_TemperatureHotWater                               :FB_BA_Label:=( sObjName:='TWW', sDescr:='Temperatur Warmwasser');
  LblAggregates_TemperatureCirculation                            :FB_BA_Label:=( sObjName:='TWZ', sDescr:='Temperatur Zirkulation');
  LblAggregates_TemperatureRecirculatingAir                       :FB_BA_Label:=( sObjName:='TUM', sDescr:='Umlufttemperatur');
  LblAggregates_TemperatureFlow                                   :FB_BA_Label:=( sObjName:='TVL', sDescr:='Vorlauftemperatur');
  LblAggregates_TemperatureSupplyAir                              :FB_BA_Label:=( sObjName:='TZU', sDescr:='Zulufttemperatur');
//481 GA-Sensorik – Druck
  LblAggregates_PressureExtractAir                                :FB_BA_Label:=( sObjName:='PAB', sDescr:='Abluftdruck');
  LblAggregates_PressureOutsideAir                                :FB_BA_Label:=( sObjName:='PAU', sDescr:='Außenluftdruck');
  LblAggregates_PressureDifferential                              :FB_BA_Label:=( sObjName:='PDI', sDescr:='Differenzdruck');
  LblAggregates_PressureDifferentialOutsideAirFilter              :FB_BA_Label:=( sObjName:='PDI', sDescr:='Differenzdruck Außenluftfilter');
  LblAggregates_PressureDifferentialExtractAirFilter              :FB_BA_Label:=( sObjName:='PDI', sDescr:='Differenzdruck Abluftfilter');
  LblAggregates_PressureDifferentialExhaustAirFilter              :FB_BA_Label:=( sObjName:='PDI', sDescr:='Differenzdruck Fortluftfilter');
  LblAggregates_PressureDifferentialSupplyAirFan                  :FB_BA_Label:=( sObjName:='PDI', sDescr:='Differenzdruck Zuluftventilator');
  LblAggregates_PressureDifferentialExtractAirFan                 :FB_BA_Label:=( sObjName:='PDI', sDescr:='Differenzdruck Abluftventilator');
  LblAggregates_PressureDifferentialExhaustAirFan                 :FB_BA_Label:=( sObjName:='PDI', sDescr:='Differenzdruck Fortluftventilator');
  LblAggregates_PressureSensorFlow                                :FB_BA_Label:=( sObjName:='PVL', sDescr:='Drucksensor (Wasser) Vorlauf');
  LblAggregates_MonitorPressure                                   :FB_BA_Label:=( sObjName:='DRW', sDescr:='Druckwächter');
  LblAggregates_PressureExhaustAir                                :FB_BA_Label:=( sObjName:='PFO', sDescr:='Fortluftdruck');
  LblAggregates_PressureRoomAir                                   :FB_BA_Label:=( sObjName:='PRU', sDescr:='Raumdruck');
  LblAggregates_PressureIndexCircuitSensorDifferential            :FB_BA_Label:=( sObjName:='PSI', sDescr:='Schlechtpunktfühler Differenzdruck');
  LblAggregates_LimiterSafetyPressure                             :FB_BA_Label:=( sObjName:='SDB', sDescr:='Sicherheitsdruckbegrenzer');
  LblAggregates_PressureSupplyAir                                 :FB_BA_Label:=( sObjName:='PZU', sDescr:='Zuluftdruck');
//481 GA-Sensorik – Luftqualität
  LblAggregates_CO2Sensor                                         :FB_BA_Label:=( sObjName:='COM', sDescr:='CO2-Sensor');
  LblAggregates_QualityExtractAir                                 :FB_BA_Label:=( sObjName:='QAB', sDescr:='Luftqualität Abluft');
  LblAggregates_OualityRoomAir                                    :FB_BA_Label:=( sObjName:='QRU', sDescr:='Luftqualität Raum');
  LblAggregates_QualitiySupplyAir                                 :FB_BA_Label:=( sObjName:='QZU', sDescr:='Luftqualität Zuluft');
  LblAggregates_QualityAirSensor                                  :FB_BA_Label:=( sObjName:='LQF', sDescr:='Luftqualitätsfühler');
//481 GA-Sensorik – Feuchte
  LblAggregates_Hygrostat                                         :FB_BA_Label:=( sObjName:='HYG', sDescr:='Hygrostat');
  LblAggregates_RelativeHumiditiyExtractAir                       :FB_BA_Label:=( sObjName:='MAB', sDescr:='Abluftfeuchte relativ');
  LblAggregates_RelativeHumidityOutsideAir                        :FB_BA_Label:=( sObjName:='MAU', sDescr:='Außenfeuchte relativ');
  LblAggregates_RelativeHumidityExhaustAir                        :FB_BA_Label:=( sObjName:='MFO', sDescr:='Fortluftfeuchte relativ');
  LblAggregates_MonitorCondensation                               :FB_BA_Label:=( sObjName:='MKW', sDescr:='Kondensationswächter');
  LblAggregates_RelativeHumidityMixedAir                          :FB_BA_Label:=( sObjName:='MMI', sDescr:='Mischluftfeuchte relativ');
  LblAggregates_RelativeHumidityRoomHumidity                      :FB_BA_Label:=( sObjName:='MRU', sDescr:='Raumfeuchte relativ');
  LblAggregates_RelativeHumidityRecirculatedAir                   :FB_BA_Label:=( sObjName:='MUM', sDescr:='Umluftfeuchte relativ');
  LblAggregates_RelativeHumiditySupplyAir                         :FB_BA_Label:=( sObjName:='MZU', sDescr:='Zuluftfeuchte relativ');
  LblAggregates_AbsoluteHumidityExtractAir                        :FB_BA_Label:=( sObjName:='XAB', sDescr:='Abluftfeuchte absolut');
  LblAggregates_AbsoluteHumidtiyOutsideAir                        :FB_BA_Label:=( sObjName:='XAU', sDescr:='Außenluftfeuchte absolut');
  LblAggregates_AbsoluteHumidtiyExhaustAir                        :FB_BA_Label:=( sObjName:='XFO', sDescr:='Fortluftfeuchte absolut');
  LblAggregates_AbsoluteHumidityMixedAir                          :FB_BA_Label:=( sObjName:='XMI', sDescr:='Mischluftfeuchte absolut');
  LblAggregates_AbsoluteHumidityRoomAir                           :FB_BA_Label:=( sObjName:='XRU', sDescr:='Raumfeuchte absolut');
  LblAggregates_AbsoluteHumidityRecirculatingAir                  :FB_BA_Label:=( sObjName:='XUM', sDescr:='Umluftfeuchte absolut');
  LblAggregates_AbsoluteHumiditySupplyAir                         :FB_BA_Label:=( sObjName:='XZU', sDescr:='Zuluftfeuchte absolut');
//481 GA-Sensorik – Verbrauchserfassung
  LblAggregates_MeterElectric                                     :FB_BA_Label:=( sObjName:='ELZ', sDescr:='Elektrozähler');
  LblAggregates_MeterGasNaturalGas                                :FB_BA_Label:=( sObjName:='EGZ', sDescr:='Gaszähler Erdgas');
  LblAggregates_MeterCoolingEnergy                                :FB_BA_Label:=( sObjName:='KMZ', sDescr:='Kältemengenzähler');
  LblAggregates_MeterHeat                                         :FB_BA_Label:=( sObjName:='WMZ', sDescr:='Wärmemengenzähler');
  LblAggregates_MetferWater                                       :FB_BA_Label:=( sObjName:='WAZ', sDescr:='Wasserzähler');
  LblAggregates_MeterFuel                                         :FB_BA_Label:=( sObjName:='BSZ', sDescr:='Brennstoffzähler (Öl)');
  LblAggregates_MeterSteam                                        :FB_BA_Label:=( sObjName:='DMZ', sDescr:='Dampfmengenzähler');
  LblAggregates_DegreeDayNumber                                   :FB_BA_Label:=( sObjName:='GTZ', sDescr:='Gradtagszahl');
//481 GA-Sensorik – Zustandserfassung und sonstige
  LblAggregates_LeakageMonitoring                                 :FB_BA_Label:=( sObjName:='LCK', sDescr:='Leckageüberwachung');
  LblAggregates_EmergencyStop                                     :FB_BA_Label:=( sObjName:='NOT', sDescr:='Not-Aus-Einrichtung/-Taster');
  LblAggregates_StockLevel                                        :FB_BA_Label:=( sObjName:='LSP', sDescr:='Speicherfüllstand');
  LblAggregates_FlowMonitor                                       :FB_BA_Label:=( sObjName:='SSW', sDescr:='Strömungswächter');
  LblAggregates_OverflowMonitoring                                :FB_BA_Label:=( sObjName:='UBL', sDescr:='Überlaufüberwachung');
  LblAggregates_LowWaterCutOff                                    :FB_BA_Label:=( sObjName:='WMS', sDescr:='Wassermangelsicherung');
  LblAggregates_WaterFlowMonitor                                  :FB_BA_Label:=( sObjName:='WSW', sDescr:='Wasserströmungswächter');
//481 GA-Sensorik – Drehzahl
  LblAggregates_PumpSpeed                                         :FB_BA_Label:=( sObjName:='SPP', sDescr:='Drehzahl Pumpe');
  LblAggregates_FanSpeedExtractAir                                :FB_BA_Label:=( sObjName:='SAB', sDescr:='Drehzahl Ventilator (Abluft)');
  LblAggregates_FanSpeedExhaustAir                                :FB_BA_Label:=( sObjName:='SFO', sDescr:='Drehzahl Ventilator (Fortluft)');
  LblAggregates_FanSpeedSupplyAir                                 :FB_BA_Label:=( sObjName:='SZU', sDescr:='Drehzahl Ventilator (Zuluft)');
//481 GA-Sensorik – Volumenstrom
  LblAggregates_VolumeFlowRateExtractAir                          :FB_BA_Label:=( sObjName:='VAB', sDescr:='Volumenstrom Abluft');
  LblAggregates_VolumeFlowRateOutsideAir                          :FB_BA_Label:=( sObjName:='VAU', sDescr:='Volumenstrom Außenluft');
  LblAggregates_VolumeFlowRateExhaustAir                          :FB_BA_Label:=( sObjName:='VFO', sDescr:='Volumenstrom Fortluft');
  LblAggregates_VolumeFlowRateBrineCirculatorySystem              :FB_BA_Label:=( sObjName:='VSO', sDescr:='Volumenstrom Sole (KVS)');
  LblAggregates_VolumeFlowRateColdDrinkingWater                   :FB_BA_Label:=( sObjName:='VKW', sDescr:='Volumenstrom Trinkwasser kalt');
  LblAggregates_VolumeFlowRateHotDrinkingWater                    :FB_BA_Label:=( sObjName:='VWW', sDescr:='Volumenstrom Trinkwasser warm');
  LblAggregates_VolumeFlowRateWaterPurification                   :FB_BA_Label:=( sObjName:='VAW', sDescr:='Volumenstrom Wasseraufbereitung');
  LblAggregates_VolumeFlowRateSupplyAir                           :FB_BA_Label:=( sObjName:='VZU', sDescr:='Volumenstrom Zuluft');
//481 GA-Aktorik – Stellantriebe
  LblAggregates_ValveRadiator                                     :FB_BA_Label:=( sObjName:='HKV', sDescr:='Heizkörperventil-Antrieb');
  LblAggregates_ValveCoolingCeiling                               :FB_BA_Label:=( sObjName:='KDV', sDescr:='Kühldeckenventil-Antrieb');
  LblAggregates_MotorisedFlap                                     :FB_BA_Label:=( sObjName:='KLA', sDescr:='Motorische Klappe');
  LblAggregates_Valve                                             :FB_BA_Label:=( sObjName:='VEN', sDescr:='Motorventil ');
  LblAggregates_HumidifierValve                                   :FB_BA_Label:=( sObjName:='VEN', sDescr:='Befeuchter Ventil ');
//481 GA-Beleuchtung
  LblAggregates_IlluminationExternal                              :FB_BA_Label:=( sObjName:='EAU', sDescr:='Beleuchtungsstärke Außen');
  LblAggregates_IlluminationRoom                                  :FB_BA_Label:=( sObjName:='ERU', sDescr:='Beleuchtungsstärke Raum');
  LblAggregates_LightColourRoom                                   :FB_BA_Label:=( sObjName:='CRU', sDescr:='Lichtfarbe Raum');
  LblAggregates_RedLightIntensity                                 :FB_BA_Label:=( sObjName:='LRT', sDescr:='Lichtintensität rot');
  LblAggregates_GreenLightIntensity                               :FB_BA_Label:=( sObjName:='LGN', sDescr:='Lichtintensität grün');
  LblAggregates_BlueLightIntensity                                :FB_BA_Label:=( sObjName:='LBL', sDescr:='Lichtintensität blau');
//481 GA-Sonnenschutz
  LblAggregates_BlindAnglePosition                                :FB_BA_Label:=( sObjName:='JWI', sDescr:='Winkelposition Jalousie');
  LblAggregates_ShadingPosition                                   :FB_BA_Label:=( sObjName:='JPO', sDescr:='Verschattungsposition');
  LblAggregates_MovementCommand                                   :FB_BA_Label:=( sObjName:='JFB', sDescr:='Jalousie Fahrbefehl');
//485 Raumautomation
  LblAggregates_DisplayAndControlUnit                             :FB_BA_Label:=( sObjName:='ABE', sDescr:='Anzeige- und Bedieneinrichtung');
  LblAggregates_PresenceSwitches                                  :FB_BA_Label:=( sObjName:='PME', sDescr:='Präsenzschalter, -melder, Bewegungsmelder');
  LblAggregates_RoomAutomationDevice                              :FB_BA_Label:=( sObjName:='RAE', sDescr:='Raumautomationseinrichtung');
  LblAggregates_RoomControlUnit                                   :FB_BA_Label:=( sObjName:='RBG', sDescr:='Raumbediengerät');
END_VAR

// ---- Templates/GVLs/DPAD/Labels/1031/LblControl1031.TcGVL
{region '#Template'}
	{attribute 'Version' := '1.0.0.0'}
	{attribute 'Tags' := '"LCID": "1031", "Text": "GVL, AKS, Labels, ObjectName, Description"'}
	{attribute 'Tags' := '"LCID": "1033", "Text": "GVL, DPAD, Labels, ObjectName, Description"'}
	{attribute 'Description' := '"LCID": "1031", "Text": "Anlagenkennzeichnungssystem, Labels controls"'}
	{attribute 'Description' := '"LCID": "1033", "Text": "Data Point Addressing Description, Labels controls"'}
{endregion}

{attribute 'global_init_slot' := '40510'}
VAR_GLOBAL
  LblControl_OperationMode                                     :FB_BA_Label:=( sObjName:='BTA', sDescr:='Betriebsart');
  LblControl_SummerNightCooling                                :FB_BA_Label:=( sObjName:='SNK', sDescr:='Sommernachtkühlung');
  LblControl_DifferencePressureMonitoringSupplyAirFan          :FB_BA_Label:=( sObjName:='DRW', sDescr:='Zuluftventilator Differenzdrucküberwachung ');
  LblControl_DifferencePressureMonitoringExtractAirFan         :FB_BA_Label:=( sObjName:='DRW', sDescr:='Abluftventilator Differenzdrucküberwachung ');
  LblControl_TSetpointCalculation                              :FB_BA_Label:=( sObjName:='SWC', sDescr:='Sollwertberechnung Temperatur');
  LblControl_HSetpointCalculation                              :FB_BA_Label:=( sObjName:='SWC', sDescr:='Sollwertberechnung Feuchte');
  LblControl_TCascadeSupplyAirControl                          :FB_BA_Label:=( sObjName:='RGL', sDescr:='Führungsregelung Zulufttemperatur');
  LblControl_HCascadeSupplyAirControl                          :FB_BA_Label:=( sObjName:='RGL', sDescr:='Führungsregelung Zuluftfeuchte');
  LblControl_PreHeater                                         :FB_BA_Label:=( sObjName:='VEH', sDescr:='Vorerhitzer');
  LblControl_ReHeater                                          :FB_BA_Label:=( sObjName:='NEH', sDescr:='Nacherhitzer');
  LblControl_EnergyRecovery                                    :FB_BA_Label:=( sObjName:='ERG', sDescr:='Energierückgewinnung');
  LblControl_SupplyAirTemperatureControl                       :FB_BA_Label:=( sObjName:='RGL', sDescr:='Zulufttemperaturregelung');
  LblControl_SupplyAirDehumidifierControl                      :FB_BA_Label:=( sObjName:='RGL', sDescr:='Zuluftentfeuchtereglung');
  LblControl_SupplyAirHumidifierController                     :FB_BA_Label:=( sObjName:='RGL', sDescr:='Zuluftfeuchtereglung');
  LblControl_SupplyAirTemperatureLimitationControl             :FB_BA_Label:=( sObjName:='RGL', sDescr:='Zulufttemperatur Begrenzungsregelung ');
  LblControl_ReturnWaterControl                                :FB_BA_Label:=( sObjName:='RGL', sDescr:='Rücklauftemperaturregelung');
  LblControl_HumidityLimitationControl                         :FB_BA_Label:=( sObjName:='RGL', sDescr:='Rel Feuchte Begrenzungsregelung');
  LblControl_CalculationPreRinseSetpoint                       :FB_BA_Label:=( sObjName:='SWB', sDescr:='Berechung Vorspülsollwert ');
  LblControl_FrostProtectionControl                            :FB_BA_Label:=( sObjName:='FSR', sDescr:='Frostschutzregelung luftseitig');
  LblControl_ExhaustAirTemperatureControl                      :FB_BA_Label:=( sObjName:='RGL', sDescr:='Fortlufttemperaturregelung');
  LblControl_EnergyRecoveryDeicingRamp                         :FB_BA_Label:=( sObjName:='RMP', sDescr:='Rampe Enteisung');
  LblControl_BACnetDevice                                      :FB_BA_Label:=( sObjName:='DEV', sDescr:='BACnet device');
  LblControl_PlantControl                                      :FB_BA_Label:=( sObjName:='ALS', sDescr:='Anlagensteuerung');
  LblControl_TSequenceControl                                  :FB_BA_Label:=( sObjName:='SEQ', sDescr:='Sequenzsteuerung Temp');
  LblControl_HSequenceControl                                  :FB_BA_Label:=( sObjName:='SEQ', sDescr:='Sequenzsteuerung Feuchte');
  LblControl_GeneralBeckhoffEventClass                         :FB_BA_Label:=( sObjName:='EKL', sDescr:='Ereignisklasse');
  LblControl_GeneralSettings                                   :FB_BA_Label:=( sObjName:='ALP', sDescr:='Anlagenparameter');
  LblControl_GeneralCabinetBasicEquipment                      :FB_BA_Label:=( sObjName:='SSG', sDescr:='Schaltschrank Grundausstattung');
  LblControl_GeneralCabinetAdditionalEquipment                 :FB_BA_Label:=( sObjName:='SSZ', sDescr:='Schaltschrank Zusatzausstattung');
  LblControl_EventIndicationLamp                               :FB_BA_Label:=( sObjName:='SMM', sDescr:='Sammelstörmeldung Lampe');
  LblControl_AcknowledgeCommand                                :FB_BA_Label:=( sObjName:='QUI', sDescr:='Hardware quittieren');
  LblControl_RemoteAcknowledgement                             :FB_BA_Label:=( sObjName:='QUI', sDescr:='Fernquittierung Störung');
  LblControl_LocalAcknowledgement                              :FB_BA_Label:=( sObjName:='QUI', sDescr:='Lokale Quittierung Störung');
  LblControl_Acknowledge                                       :FB_BA_Label:=( sObjName:='QUI', sDescr:='Quittierung');
// 
  LblControl_Fuse                                              :FB_BA_Label:=( sObjName:='SIC', sDescr:='Sicherung');
// Einstellungen
  LblControl_FrostProtection                                   :FB_BA_Label:=( sObjName:='FRS', sDescr:='Frostschutz');
  LblControl_MinimumOutsideTemperature                         :FB_BA_Label:=( sObjName:='TWI', sDescr:='Minimale Außentemperatur');
  LblControl_TemperatureWeatherLowLimit                        :FB_BA_Label:=( sObjName:='TWI', sDescr:='Minimale Außentemperatur unterer Grenzwert');
  LblControl_TemperatureWeatherDamped                          :FB_BA_Label:=( sObjName:='TWG', sDescr:='Temperatur Witterung gedämpft');
  LblControl_TemperatureWeatherDampedLowLimit                  :FB_BA_Label:=( sObjName:='TWG', sDescr:='Temperatur Witterung gedämpft unterer Grenzwert');
  LblControl_PressureControl                                   :FB_BA_Label:=( sObjName:='RGL', sDescr:='Druckregelung');
  LblControl_Converter3Point                                   :FB_BA_Label:=( sObjName:='WDL', sDescr:='3 Punkt Wandler');
  LblControl_HeatingCurve                                      :FB_BA_Label:=( sObjName:='HKV', sDescr:='Heizkurve');
  LblControl_SetpointGeneration                                :FB_BA_Label:=( sObjName:='SWG', sDescr:='Sollwert Generierung');
  LblControl_RequestHeatState                                  :FB_BA_Label:=( sObjName:='AWZ', sDescr:='Wärmeanforderung Zustand');
  LblControl_RequestHeatSetpoint                               :FB_BA_Label:=( sObjName:='AWS', sDescr:='Wärmeanforderung Sollwert');
  LblControl_FlowTempControl                                   :FB_BA_Label:=( sObjName:='RGL', sDescr:='Vorlauf Temperatur Regelung');
// 
  LblControl_RoomTemperatureControl                            :FB_BA_Label:=( sObjName:='RGL', sDescr:='Raumtemperaturregelung');
  LblControl_FlowTemperatureControl                            :FB_BA_Label:=( sObjName:='RGL', sDescr:='Vorlauftemperatur Regelung');
  LblControl_SetpointHeating                                   :FB_BA_Label:=( sObjName:='SWG', sDescr:='Sollwertgenerierung heizen');
  LblControl_SetpointCooling                                   :FB_BA_Label:=( sObjName:='SWG', sDescr:='Sollwertgenerierung kühlen');
  LblControl_Facade                                            :FB_BA_Label:=( sObjName:='FEE', sDescr:='Fassadendaten');
  LblControl_BuildingAlarms                                    :FB_BA_Label:=( sObjName:='FEE', sDescr:='Gebäude Alarme');
  LblControl_BuildingEnergyLevel                               :FB_BA_Label:=( sObjName:='FEE', sDescr:='Gebäude Energieniveaus');
  LblControl_BuildingMode                                      :FB_BA_Label:=( sObjName:='FEE', sDescr:='Gebäude Betriebsmodus');
  LblControl_BuildingSpRmT                                     :FB_BA_Label:=( sObjName:='FEE', sDescr:='Gebäude Raumtemperatursollwerte');
  LblControl_BuildingSunprotection                             :FB_BA_Label:=( sObjName:='FEE', sDescr:='Gebäude Sonnenschutz');
  LblControl_TemperatureFrost                                  :FB_BA_Label:=( sObjName:='TFR', sDescr:='Temperatur Frost');
  LblControl_MixedAirStartUpRamp                               :FB_BA_Label:=( sObjName:='RMP', sDescr:='Rampe Anlagenstart');
  LblControl_Cooler                                            :FB_BA_Label:=( sObjName:='KUE', sDescr:='Kühler');
  LblControl_EvtCategoryLifeSafty                              :FB_BA_Label:=( sObjName:='EKL', sDescr:='Lebensgefahr');
  LblControl_EvtCategoryAlarmTechnical                         :FB_BA_Label:=( sObjName:='EKT', sDescr:='Techn Alarm');
  LblControl_EvtCategoryDisturbance                            :FB_BA_Label:=( sObjName:='EKS', sDescr:='Störung');
  LblControl_EvtCategoryMaintenance                            :FB_BA_Label:=( sObjName:='EKW', sDescr:='Wartung');
  LblControl_EvtCategoryNotification                           :FB_BA_Label:=( sObjName:='EKB', sDescr:='Benachrichtigung ');
  LblControl_EvtCategoryOther                                  :FB_BA_Label:=( sObjName:='EKA', sDescr:='Sonstiges');
  LblControl_TrendLogging                                      :FB_BA_Label:=( sObjName:='TRA', sDescr:='Trend ');
  LblControl_WeatherParameters                                 :FB_BA_Label:=( sObjName:='PWI', sDescr:='Witterung Parameter');
  LblControl_SetpointFrostProtection                           :FB_BA_Label:=( sObjName:='SW_', sDescr:='Sollwert Frostschutz');
  LblControl_SetpointWeatherIcing                              :FB_BA_Label:=( sObjName:='SW_', sDescr:='Sollwert Vereisung');
  LblControl_SetpointMinimumOutsideTemperature                 :FB_BA_Label:=( sObjName:='SWI', sDescr:='Sollwert Minimale Außentemperatur');
  LblControl_MeanDamped                                        :FB_BA_Label:=( sObjName:='MWT', sDescr:='Mittelwert Außentemperatur gedämpft');
  LblControl_OperationalMessageTemperatureWeatherLowLimit      :FB_BA_Label:=( sObjName:='BM_', sDescr:='Betriebsmeldung Außentemperatur unterer Grenzwert');
  LblControl_OperationalMessageTemperatureWeatherDampedLowLimit:FB_BA_Label:=( sObjName:='BM_', sDescr:='Betriebsmeldung Außentemperatur gedämpft unterer Grenzwert');
// Beckhoff Schaltschrank Grundausstattung
  LblControl_SwitchingCommandCollectiveFaultSignalLamp         :FB_BA_Label:=( sObjName:='SB_', sDescr:='Sammelstörmeldung Lampe Schaltbefehl');
  LblControl_SwitchingCommandHardwareAcknowledgement           :FB_BA_Label:=( sObjName:='SB_', sDescr:='Hardware quittieren Schaltbefehl');
  LblControl_ButtonRemoteAcknowledgement                       :FB_BA_Label:=( sObjName:='TS_', sDescr:='Eingabe Fernquittierung');
  LblControl_ButtonLocalAcknowledgement                        :FB_BA_Label:=( sObjName:='TS_', sDescr:='Taster Quittierung');
// Beckhoff Heizkreis
  LblControl_HeatingLimit                                      :FB_BA_Label:=( sObjName:='HGW', sDescr:='Heizgrenzwert');
  LblControl_PresentOperationMode                              :FB_BA_Label:=( sObjName:='ABA', sDescr:='aktuelle Betriebsart');
  LblControl_OperationModeSelection                            :FB_BA_Label:=( sObjName:='BAA', sDescr:='Betriebsartenauswahl');
// Beckhoff Sommernachtkühlung
  LblControl_HysteresisRoomTemperature                         :FB_BA_Label:=( sObjName:='HYS', sDescr:='Hysterese Raumtemperatur');
  LblControl_OutsideTemperatureLowLimit                        :FB_BA_Label:=( sObjName:='MIN', sDescr:='minimale Außentemperatur');
  LblControl_OffValueDifferenceOutsideInsightTemperature       :FB_BA_Label:=( sObjName:='MIN', sDescr:='Ausschaltwert von Differenz Außentemperatur - Raumtemperatur');
  LblControl_OnValueDifferenceOutsideInsightTemperature        :FB_BA_Label:=( sObjName:='MAX', sDescr:='Einschaltwert von Differenz Außentemperatur - Raumtemperatur');
// Beckhoff Klappen
  LblControl_DriveTimeOpen                                     :FB_BA_Label:=( sObjName:='LZA', sDescr:='Laufzeit Auf');
  LblControl_DriveTimeClose                                    :FB_BA_Label:=( sObjName:='LZZ', sDescr:='Laufzeit Zu ');
  LblControl_DisturbanceFeedbackOpen                           :FB_BA_Label:=( sObjName:='SMA', sDescr:='Störung Rückmeldung Auf');
  LblControl_DisturbanceFeedbackClose                          :FB_BA_Label:=( sObjName:='SMZ', sDescr:='Störung Rückmeldung Zu');
// Beckhoff Differenzdrucküberwachung
  LblControl_TimeDelay                                         :FB_BA_Label:=( sObjName:='ZV_', sDescr:='Verzögerung ');
  LblControl_TimeDelayFeedback                                 :FB_BA_Label:=( sObjName:='ZVR', sDescr:='Verzögerung Rückmeldung');
  LblControl_TimeDelayInterruptionFeedback                     :FB_BA_Label:=( sObjName:='ANV', sDescr:='Ansprechverzögerung ');
// Beckhoff Vorspülen
  LblControl_PreRinseDuration                                  :FB_BA_Label:=( sObjName:='VSP', sDescr:='Vorspüldauer');
  LblControl_DisturbancePreRinse                               :FB_BA_Label:=( sObjName:='SM_', sDescr:='Meldung Störung Vorspülen');
  LblControl_SetpointMinimalReturnWaterTemperature             :FB_BA_Label:=( sObjName:='SW_', sDescr:='Sollwert minimale Rücklauftemperatur');
// Beckhoff  Rampe
  LblControl_RampTimeUp                                        :FB_BA_Label:=( sObjName:='RPA', sDescr:='Rampenzeit auf');
  LblControl_RampTimeDown                                      :FB_BA_Label:=( sObjName:='RPZ', sDescr:='Rampenzeit ab');
  LblControl_CommandOpen                                       :FB_BA_Label:=( sObjName:='SB_', sDescr:='Schaltbefehl Auf');
  LblControl_CommandClose                                      :FB_BA_Label:=( sObjName:='SB_', sDescr:='Schaltbefehl Zu');
  LblControl_CalculatedValue                                   :FB_BA_Label:=( sObjName:='ERW', sDescr:='errechneter Wert');
  LblControl_Value                                             :FB_BA_Label:=( sObjName:='WET', sDescr:='Wert');
// Beckhoff Ereignisklassen
  LblControl_EvtClassSimple                                    :FB_BA_Label:=( sObjName:='NC_', sDescr:='Einfach');
  LblControl_EvtClassStandard                                  :FB_BA_Label:=( sObjName:='NC_', sDescr:='Standard');
  LblControl_EvtClassExtended                                  :FB_BA_Label:=( sObjName:='NC_', sDescr:='Erweitert');
  LblControl_FlowSwitch                                        :FB_BA_Label:=( sObjName:='BM_', sDescr:='Betriebsmeldung Strömungswächter');
  LblControl_SmokeAlarm                                        :FB_BA_Label:=( sObjName:='SM_', sDescr:='Störung Rauchalarm');
  LblControl_SystemFailure                                     :FB_BA_Label:=( sObjName:='SM_', sDescr:='Störung Systemfehler');
  LblControl_Contamination                                     :FB_BA_Label:=( sObjName:='SM_', sDescr:='Störung Kontamination');
  LblControl_SwitchingCommandSmokeDetector                     :FB_BA_Label:=( sObjName:='SB_', sDescr:='Schaltbefehl Quittierung');
  LblControl_ButtonReset                                       :FB_BA_Label:=( sObjName:='TS_', sDescr:='Taster Quittierung');
  LblControl_OffsetNightSetpoint                               :FB_BA_Label:=( sObjName:='SNK', sDescr:='Offset Nachtabsenkung');
// 
  LblControl_SetpointRelHumidityHumidification                 :FB_BA_Label:=( sObjName:='SW_', sDescr:='Sollwert Relative Feuchte Befeuchten');
  LblControl_SetpointRelHumidityDehumidification               :FB_BA_Label:=( sObjName:='SW_', sDescr:='Sollwert Relative Feuchte Entfeuchten');
  LblControl_SetpointAbsHumidityHumidification                 :FB_BA_Label:=( sObjName:='SWC', sDescr:='Sollwert Absolute Feuchte Befeuchten');
  LblControl_SetpointAbsHumidityDehumidification               :FB_BA_Label:=( sObjName:='SWC', sDescr:='Sollwert Absolute Feuchte Entfeuchten');
  LblControl_SetpointRelHumidity                               :FB_BA_Label:=( sObjName:='SW_', sDescr:='Sollwert Relative Feuchte');
  LblControl_SetpointAbsHumidity                               :FB_BA_Label:=( sObjName:='SW_', sDescr:='Sollwert Absolute Feuchte');
  LblControl_OperationalMessageDehumidification                :FB_BA_Label:=( sObjName:='BM_', sDescr:='Betriebsmeldung Entfeuchtung');
// 
  LblControl_SetpointSunblindPosition                          :FB_BA_Label:=( sObjName:='SW_', sDescr:='Sollwert Jalousie Position');
  LblControl_SetpointSunblindAngle                             :FB_BA_Label:=( sObjName:='SW_', sDescr:='Sollwert Jalousie Winkel');
  LblControl_CommandSunblindStart                              :FB_BA_Label:=( sObjName:='SB_', sDescr:='Startbefehl');
  LblControl_ButtonSunblind                                    :FB_BA_Label:=( sObjName:='TS_', sDescr:='Jalousietaster');
  LblControl_FeedbackSunblindPosition                          :FB_BA_Label:=( sObjName:='RM_', sDescr:='Rückmeldung Jalousie Position');
  LblControl_FeedbackSunblindAngle                             :FB_BA_Label:=( sObjName:='RM_', sDescr:='Rückmeldung Jalousie Winkel');
  LblControl_FeedbackSunblindPrio                              :FB_BA_Label:=( sObjName:='RM_', sDescr:='Rückmeldung Telegrammpriorität');
// 
  LblControl_TimeDelayStormOn                                  :FB_BA_Label:=( sObjName:='ESV', sDescr:='Sturmerkennung Verzögerung Ein');
  LblControl_TimeDelayStormOff                                 :FB_BA_Label:=( sObjName:='ASV', sDescr:='Sturmerkennung Verzögerung Aus');
  LblControl_MaintenanceEnable                                 :FB_BA_Label:=( sObjName:='FRG', sDescr:='Wartungsposition Freigabe');
  LblControl_MaintenancePosition                               :FB_BA_Label:=( sObjName:='SW_', sDescr:='Sollwert Wartung Position');
  LblControl_MaintenanceAngle                                  :FB_BA_Label:=( sObjName:='SW_', sDescr:='Sollwert Wartung Winkel');
  LblControl_FacadeThermoAutomaticEnable                       :FB_BA_Label:=( sObjName:='FRG', sDescr:='Fassaden-Thermoautomatik Freigabe');
  LblControl_FacadeThermoAutomaticCoolingPosition              :FB_BA_Label:=( sObjName:='SW_', sDescr:='Fassaden-Thermoautomatik Kühl-Position');
  LblControl_FacadeThermoAutomaticCoolingAngle                 :FB_BA_Label:=( sObjName:='SW_', sDescr:='Fassaden-Thermoautomatik Kühl-Winkel');
  LblControl_FacadeTwilightAutomaticEnable                     :FB_BA_Label:=( sObjName:='FRG', sDescr:='Fassaden-Dämmerungsautomatik Freigabe');
  LblControl_SunProtectionValueOn                              :FB_BA_Label:=( sObjName:='SW_', sDescr:='Sonnenschutz Helligkeitswert Ein');
  LblControl_SunProtectionValueOff                             :FB_BA_Label:=( sObjName:='SW_', sDescr:='Sonnenschutz Helligkeitswert Aus');
  LblControl_TimeDelaySunProtectionOn                          :FB_BA_Label:=( sObjName:='ESV', sDescr:='Sonnenschutz Verzögerung Ein');
  LblControl_TimeDelaySunProtectionOff                         :FB_BA_Label:=( sObjName:='ASV', sDescr:='Sonnenschutz Verzögerung Aus');
  LblControl_FacadeParkingEnable                               :FB_BA_Label:=( sObjName:='FRG', sDescr:='Fassaden-Parken Freigabe');
  LblControl_FacadeParkingPosition                             :FB_BA_Label:=( sObjName:='SW_', sDescr:='Fassaden-Parken Position');
  LblControl_FacadeParkingAngle                                :FB_BA_Label:=( sObjName:='SW_', sDescr:='Fassaden-Parken Winkel');
  LblControl_WindProtectionState                               :FB_BA_Label:=( sObjName:='STA', sDescr:='Status Sturmschutz');
  LblControl_SunProtectionState                                :FB_BA_Label:=( sObjName:='STA', sDescr:='Status Sonnenschutz');
// 
  LblControl_LowWaterMonitor                                   :FB_BA_Label:=( sObjName:='SM_', sDescr:='Wassermangelwächter');
  LblControl_FireAlert                                         :FB_BA_Label:=( sObjName:='SM_', sDescr:='Feueralarm');
  LblControl_Burglary                                          :FB_BA_Label:=( sObjName:='SM_', sDescr:='Einbruchalarm');
  LblControl_CentralSwitchOff                                  :FB_BA_Label:=( sObjName:='ALS', sDescr:='Zentraler Schalter Aus');
  LblControl_ForcedVentilation                                 :FB_BA_Label:=( sObjName:='ALS', sDescr:='Zwangsbelüftung');
  LblControl_SmokeExtraction                                   :FB_BA_Label:=( sObjName:='ALS', sDescr:='Entrauchung');
  LblControl_SetpointIce                                       :FB_BA_Label:=( sObjName:='SW_', sDescr:='Vereisungstemperatur');
  LblControl_SunProtectionInterval                             :FB_BA_Label:=( sObjName:='SW_', sDescr:='Sonnenschutz Positionierintervall');
  LblControl_DeiceTime                                         :FB_BA_Label:=( sObjName:='SW_', sDescr:='Vereisungsschutz Enteisungszeit');
  LblControl_GlobalThermoAutomaticValueOn                      :FB_BA_Label:=( sObjName:='SW_', sDescr:='Thermoautomatik Strahlungswert Ein');
  LblControl_GlobalThermoAutomaticValueOff                     :FB_BA_Label:=( sObjName:='SW_', sDescr:='Thermoautomatik Strahlungswert Aus');
  LblControl_GlobalTwilightAutomaticValueOn                    :FB_BA_Label:=( sObjName:='SW_', sDescr:='Dämmerungsautomatik Helligkeitswertwert Ein');
  LblControl_GlobalTwilightAutomaticValueOff                   :FB_BA_Label:=( sObjName:='SW_', sDescr:='Dämmerungsautomatik Helligkeitswertwert Aus');
  LblControl_IceAlert                                          :FB_BA_Label:=( sObjName:='SM_', sDescr:='Vereisungsalarm');
  LblControl_GlobalThermoAutomaticRelease                      :FB_BA_Label:=( sObjName:='FRG', sDescr:='Thermoautomatik Freigabe');
  LblControl_GlobalTwilightAutomaticRelease                    :FB_BA_Label:=( sObjName:='FRG', sDescr:='Dämmerungsautomatik Freigabe');
  LblControl_GlobalResetManMode                                :FB_BA_Label:=( sObjName:='ALS', sDescr:='Globaler Reset Handmodus');
// 
  LblControl_BuildingEnergyLevelManual                         :FB_BA_Label:=( sObjName:='BAA', sDescr:='Gebäudeenergieniveau manuelle Auswahl');
  LblControl_BuildingEnergyLevelActual                         :FB_BA_Label:=( sObjName:='ABA', sDescr:='Gebäudeenergieniveau aktuelle Auswahl');
  LblControl_BuildingEnergyLevelSched                          :FB_BA_Label:=( sObjName:='ZPL', sDescr:='Gebäudeenergieniveau Zeitschaltplan');
  LblControl_BuildingModeManual                                :FB_BA_Label:=( sObjName:='BAA', sDescr:='Gebäudebetriebsart manuelle Auswahl');
  LblControl_BuildingModeActual                                :FB_BA_Label:=( sObjName:='ABA', sDescr:='Gebäudebetriebsart aktuelle Auswahl');
  LblControl_BuildingModeSched                                 :FB_BA_Label:=( sObjName:='ZPL', sDescr:='Gebäudebetriebsart Zeitschaltplan');
// 
  LblControl_SummerCompensationX1                              :FB_BA_Label:=( sObjName:='SPX', sDescr:='Sommerkompensation X1');
  LblControl_SummerCompensationX2                              :FB_BA_Label:=( sObjName:='SPX', sDescr:='Sommerkompensation X2');
  LblControl_SummerCompensationY1                              :FB_BA_Label:=( sObjName:='SPY', sDescr:='Sommerkompensation Y1');
  LblControl_SummerCompensationY2                              :FB_BA_Label:=( sObjName:='SPY', sDescr:='Sommerkompensation Y2');
  LblControl_WinterCompensationX1                              :FB_BA_Label:=( sObjName:='SPX', sDescr:='Winterkompensation X1');
  LblControl_WinterCompensationX2                              :FB_BA_Label:=( sObjName:='SPX', sDescr:='Winterkompensation X2');
  LblControl_WinterCompensationY1                              :FB_BA_Label:=( sObjName:='SPY', sDescr:='Winterkompensation Y1');
  LblControl_WinterCompensationY2                              :FB_BA_Label:=( sObjName:='SPY', sDescr:='Winterkompensation Y2');
  LblControl_SummerCompensation                                :FB_BA_Label:=( sObjName:='SKP', sDescr:='Sommerkompensation');
  LblControl_WinterCompensation                                :FB_BA_Label:=( sObjName:='WKP', sDescr:='Winterkompensation');
  LblControl_SummerCompensationYmin                            :FB_BA_Label:=( sObjName:='SWI', sDescr:='Sommer Kompensation Ymin');
  LblControl_SummerCompensationYmax                            :FB_BA_Label:=( sObjName:='SWX', sDescr:='Sommer Kompensation Ymax');
  LblControl_WinterCompensationYmin                            :FB_BA_Label:=( sObjName:='SWI', sDescr:='Winter Kompensation Ymin');
  LblControl_WinterCompensationYmax                            :FB_BA_Label:=( sObjName:='SWX', sDescr:='Winter Kompensation Ymax');
  LblControl_SummerCompensationSp                              :FB_BA_Label:=( sObjName:='SWC', sDescr:='Sommer Kompensation Sollwert');
  LblControl_WinterCompensationSp                              :FB_BA_Label:=( sObjName:='SWC', sDescr:='Winter Kompensation Sollwert');
  LblControl_SetpointShiftHeating                              :FB_BA_Label:=( sObjName:='SW_', sDescr:='Sollwertverschiebung Heizen');
  LblControl_SetpointShiftCooling                              :FB_BA_Label:=( sObjName:='SW_', sDescr:='Sollwertverschiebung Kühlen');
  LblControl_DampConstant                                      :FB_BA_Label:=( sObjName:='SW_', sDescr:='Dämpfungskonstante');
// 
  LblControl_DelayOn                                           :FB_BA_Label:=( sObjName:='ESV', sDescr:='Einschaltverzögerung');
  LblControl_DelayOff                                          :FB_BA_Label:=( sObjName:='ASV', sDescr:='Ausschaltverzögerung');
  LblControl_AntiBlocking                                      :FB_BA_Label:=( sObjName:='BKS', sDescr:='Blockierschutz');
  LblControl_IdlePeriod                                        :FB_BA_Label:=( sObjName:='ITV', sDescr:='Intervall');
  LblControl_ImpulsLength                                      :FB_BA_Label:=( sObjName:='IPL', sDescr:='Impulslänge');
  LblControl_SuppyAirTempSetpointHeaterCalc                    :FB_BA_Label:=( sObjName:='SWC', sDescr:='Zuluft Sw Erhitzer errechnet');
  LblControl_SuppyAirTempSetpointCoolerCalc                    :FB_BA_Label:=( sObjName:='SWC', sDescr:='Zuluft Sw Kühler errechnet');
  LblControl_SuppyAirTempSetpointERCCalc                       :FB_BA_Label:=( sObjName:='SWC', sDescr:='Zuluft Sw ERG errechnet');
  LblControl_X01                                               :FB_BA_Label:=( sObjName:='SWX', sDescr:='Wert Stützpunkt [X1]');
  LblControl_X02                                               :FB_BA_Label:=( sObjName:='SWX', sDescr:='Wert Stützpunkt [X2]');
  LblControl_X03                                               :FB_BA_Label:=( sObjName:='SWX', sDescr:='Wert Stützpunkt [X3]');
  LblControl_X04                                               :FB_BA_Label:=( sObjName:='SWX', sDescr:='Wert Stützpunkt [X4]');
  LblControl_X05                                               :FB_BA_Label:=( sObjName:='SWX', sDescr:='Wert Stützpunkt [X5]');
  LblControl_X06                                               :FB_BA_Label:=( sObjName:='SWX', sDescr:='Wert Stützpunkt [X6]');
  LblControl_X07                                               :FB_BA_Label:=( sObjName:='SWX', sDescr:='Wert Stützpunkt [X7]');
  LblControl_Y01                                               :FB_BA_Label:=( sObjName:='SWY', sDescr:='Wert Stützpunkt [Y1]');
  LblControl_Y02                                               :FB_BA_Label:=( sObjName:='SWY', sDescr:='Wert Stützpunkt [Y2]');
  LblControl_Y02_03                                            :FB_BA_Label:=( sObjName:='SWY', sDescr:='Wert Stützpunkt [Y2-Y3]');
  LblControl_Y03                                               :FB_BA_Label:=( sObjName:='SWY', sDescr:='Wert Stützpunkt [Y3]');
  LblControl_Y04                                               :FB_BA_Label:=( sObjName:='SWY', sDescr:='Wert Stützpunkt [Y4]');
  LblControl_Y05                                               :FB_BA_Label:=( sObjName:='SWY', sDescr:='Wert Stützpunkt [Y5]');
  LblControl_Y06                                               :FB_BA_Label:=( sObjName:='SWY', sDescr:='Wert Stützpunkt [Y6]');
  LblControl_Y07                                               :FB_BA_Label:=( sObjName:='SWY', sDescr:='Wert Stützpunkt [Y7]');
  LblControl_Feedback                                          :FB_BA_Label:=( sObjName:='RMW', sDescr:='Rückmeldeüberwachung');
  LblControl_PreAlarmLimitMAX                                  :FB_BA_Label:=( sObjName:='GWX', sDescr:='Voralarm Grenzwert MAX');
  LblControl_PreAlarmLimitMIN                                  :FB_BA_Label:=( sObjName:='GWI', sDescr:='Voralarm Grenzwert MIN');
  LblControl_PreAlarmFault                                     :FB_BA_Label:=( sObjName:='SM_', sDescr:='Voralarm Störung');
  LblControl_MainAlarmLimitMAX                                 :FB_BA_Label:=( sObjName:='GWX', sDescr:='Hauptalarm Grenzwert MAX');
  LblControl_MainAlarmLimitMIN                                 :FB_BA_Label:=( sObjName:='GWI', sDescr:='Hauptalarm Grenzwert MIN');
  LblControl_MainAlarmFault                                    :FB_BA_Label:=( sObjName:='SM_', sDescr:='Hauptalarm Störung');
  LblControl_ProcPreRinse                                      :FB_BA_LabelProcess:=( sProcessName:='Vorspülen');
  LblControl_ProjectInfo                                       :FB_BA_Label:=( sObjName:='PI_', sDescr:='Projektinformationen');
END_VAR

// ---- Templates/GVLs/DPAD/Labels/1031/LblFunctions1031.TcGVL
{region '#Template'}
	{attribute 'Version' := '1.0.0.0'}
	{attribute 'Tags' := '"LCID": "1031", "Text": "GVL, AKS, Labels, ObjectName, Description"'}
	{attribute 'Tags' := '"LCID": "1033", "Text": "GVL, DPAD, Labels, ObjectName, Description"'}
	{attribute 'Description' := '"LCID": "1031", "Text": "Anlagenkennzeichnungssystem, Labels functions"'}
	{attribute 'Description' := '"LCID": "1033", "Text": "Data Point Addressing Description, Labels functions"'}
{endregion}

{attribute 'global_init_slot' := '40510'}
VAR_GLOBAL
  LblFunctions_Requirement                                       :FB_BA_Label:=( sObjName:='AF_', sDescr:='Anforderung');
  LblFunctions_SystemSwitch                                      :FB_BA_Label:=( sObjName:='ALS', sDescr:='Anlagenschalter');
  LblFunctions_StatusOccupiedRoom                                :FB_BA_Label:=( sObjName:='BEL', sDescr:='Belegtzustand Raum');
  LblFunctions_LimitCalculatedValue                              :FB_BA_Label:=( sObjName:='GWC', sDescr:='Berechneter Grenzwert');
  LblFunctions_SetpointCalculated                                :FB_BA_Label:=( sObjName:='SWC', sDescr:='Berechneter Sollwert');
  LblFunctions_ReadyForOperation                                 :FB_BA_Label:=( sObjName:='BB_', sDescr:='Betriebsbereit');
  LblFunctions_OperationalMessage                                :FB_BA_Label:=( sObjName:='BM_', sDescr:='Betriebsmeldung');
  LblFunctions_HoursOfOperation                                  :FB_BA_Label:=( sObjName:='BZ_', sDescr:='Betriebsstunden');
  LblFunctions_LimitValueHoursOfOperation                        :FB_BA_Label:=( sObjName:='BZG', sDescr:='Betriebsstunden Grenzwert');
  LblFunctions_ObjectCalendar                                    :FB_BA_Label:=( sObjName:='CAL', sDescr:='Calendar-Objekt');
  LblFunctions_ObjectCommand                                     :FB_BA_Label:=( sObjName:='COM', sDescr:='Command-Objekt');
  LblFunctions_DifferentialConstantController                    :FB_BA_Label:=( sObjName:='TV_', sDescr:='Differenzialkonstante Regler');
  LblFunctions_SwitchOnErrorUnauthorisedON                       :FB_BA_Label:=( sObjName:='EF_', sDescr:='Einschaltfehler, unerlaubt EIN');
  LblFunctions_EnergyLevel                                       :FB_BA_Label:=( sObjName:='EN_', sDescr:='Energieniveau');
  LblFunctions_EnergyLevelCalculated                             :FB_BA_Label:=( sObjName:='ENC', sDescr:='Energieniveau berechnet');
  LblFunctions_UnlockingDevice                                   :FB_BA_Label:=( sObjName:='ENT', sDescr:='Entriegelung');
  LblFunctions_ObjectEventEnrollment                             :FB_BA_Label:=( sObjName:='EE_', sDescr:='Event-Enrollment-Objekt');
  LblFunctions_Enabled                                           :FB_BA_Label:=( sObjName:='FR_', sDescr:='Freigabe');
  LblFunctions_DangerAlarm                                       :FB_BA_Label:=( sObjName:='GM_', sDescr:='Gefahrmeldung');
  LblFunctions_Threshold                                         :FB_BA_Label:=( sObjName:='GW_', sDescr:='Grenzwert');
  LblFunctions_LimitMAX                                          :FB_BA_Label:=( sObjName:='GWX', sDescr:='Grenzwert MAX');
  LblFunctions_LimitMIN                                          :FB_BA_Label:=( sObjName:='GWI', sDescr:='Grenzwert MIN');
  LblFunctions_LimitNight                                        :FB_BA_Label:=( sObjName:='GWN', sDescr:='Grenzwert Nacht');
  LblFunctions_LimitDay                                          :FB_BA_Label:=( sObjName:='GWT', sDescr:='Grenzwert Tag');
  LblFunctions_ObjectGroup                                       :FB_BA_Label:=( sObjName:='GP_', sDescr:='Group-Objekt');
  LblFunctions_localPriorityAndOperatingUnitsManualMessage       :FB_BA_Label:=( sObjName:='HD_', sDescr:='LVB-Handmeldung');
  LblFunctions_HeatingCharacteristicCurveExponent                :FB_BA_Label:=( sObjName:='HEX', sDescr:='Heizkennlinie Exponent');
  LblFunctions_HeatingCharacteristicCurveParallelDisplacement    :FB_BA_Label:=( sObjName:='HPV', sDescr:='Heizkennlinie Parallelverschiebung');
  LblFunctions_HeatingCharacteristicCurveSteepness               :FB_BA_Label:=( sObjName:='HST', sDescr:='Heizkennlinie Steilheit');
  LblFunctions_HeatingCircuitNightReduction                      :FB_BA_Label:=( sObjName:='NAH', sDescr:='Heizkreis Nachtabsenkung');
  LblFunctions_Hysteresis                                        :FB_BA_Label:=( sObjName:='HYS', sDescr:='Hysterese');
  LblFunctions_Calendar                                          :FB_BA_Label:=( sObjName:='KAL', sDescr:='Kalender');
  LblFunctions_RuntimeError                                      :FB_BA_Label:=( sObjName:='LFZ', sDescr:='Laufzeitfehler');
  LblFunctions_LoopMAXLimit                                      :FB_BA_Label:=( sObjName:='LPX', sDescr:='Loop-MAX-Begrenzung');
  LblFunctions_LoopMINLimit                                      :FB_BA_Label:=( sObjName:='LPI', sDescr:='Loop-MIN-Begrenzung');
  LblFunctions_LoopObject                                        :FB_BA_Label:=( sObjName:='LP_', sDescr:='Regler');
  LblFunctions_LoopObjectCascadeSupplyAirTemperature             :FB_BA_Label:=( sObjName:='LP_', sDescr:='Führungsregler Zulufttemperatur');
  LblFunctions_LoopObjectCascadeSupplyAirHumidity                :FB_BA_Label:=( sObjName:='LP_', sDescr:='Führungsregler Zuluftfeuchte');
  LblFunctions_MaximumValue                                      :FB_BA_Label:=( sObjName:='MAX', sDescr:='Maximalwert');
  LblFunctions_MeasuredValue                                     :FB_BA_Label:=( sObjName:='MW_', sDescr:='Messwert');
  LblFunctions_MeasuredValueCalculated                           :FB_BA_Label:=( sObjName:='MWC', sDescr:='Berechneter Messwert');
  LblFunctions_MeasuredValueEast                                 :FB_BA_Label:=( sObjName:='MW_', sDescr:='Messwert Osten');
  LblFunctions_MeasuredValueNorth                                :FB_BA_Label:=( sObjName:='MW_', sDescr:='Messwert Norden');
  LblFunctions_MeasuredValueSouth                                :FB_BA_Label:=( sObjName:='MW_', sDescr:='Messwert Sueden');
  LblFunctions_MeasuredValueWest                                 :FB_BA_Label:=( sObjName:='MW_', sDescr:='Messwert Westen');
  LblFunctions_MinimumValue                                      :FB_BA_Label:=( sObjName:='MIN', sDescr:='Minimalwert');
  LblFunctions_Mean                                              :FB_BA_Label:=( sObjName:='MWT', sDescr:='Mittelwert');
  LblFunctions_FollowUpTime                                      :FB_BA_Label:=( sObjName:='NL_', sDescr:='Nachlaufzeit');
  LblFunctions_ResetTime                                         :FB_BA_Label:=( sObjName:='TN_', sDescr:='Nachstellzeit');
  LblFunctions_FeedbackDelay                                     :FB_BA_Label:=( sObjName:='ZVR', sDescr:='Zeitverzögerung Rückmeldung');
  LblFunctions_ObjectNotificationClass                           :FB_BA_Label:=( sObjName:='NC_', sDescr:='Notification-Class-Objekt');
  LblFunctions_EventClassObject                                  :FB_BA_Label:=( sObjName:='EKL', sDescr:='Ereignisklasse');
  LblFunctions_Programobject                                     :FB_BA_Label:=( sObjName:='PRG', sDescr:='Programm');
  LblFunctions_ProportionalBand                                  :FB_BA_Label:=( sObjName:='XP_', sDescr:='Proportionalband');
  LblFunctions_FeedbackOPEN                                      :FB_BA_Label:=( sObjName:='RMA', sDescr:='Rückmeldung AUF');
  LblFunctions_FeedbackCLOSED                                    :FB_BA_Label:=( sObjName:='RMZ', sDescr:='Rückmeldung ZU');
  LblFunctions_FeedbackValue                                     :FB_BA_Label:=( sObjName:='RW_', sDescr:='Rückführwert');
  LblFunctions_FeedbackErrorOPEN                                 :FB_BA_Label:=( sObjName:='RFA', sDescr:='Rückmeldefehler AUF');
  LblFunctions_FeedbackErrorCLOSED                               :FB_BA_Label:=( sObjName:='RFZ', sDescr:='Rückmeldefehler ZU');
  LblFunctions_Feedback                                          :FB_BA_Label:=( sObjName:='RM_', sDescr:='Rückmeldung');
  LblFunctions_ExecutionControl                                  :FB_BA_Label:=( sObjName:='RF_', sDescr:='Ausführkontrolle');
  LblFunctions_SwitchingCommand                                  :FB_BA_Label:=( sObjName:='SB_', sDescr:='Schaltbefehl');
  LblFunctions_Scheduler                                         :FB_BA_Label:=( sObjName:='ZPL', sDescr:='Zeitschaltplan');
  LblFunctions_Setpoint                                          :FB_BA_Label:=( sObjName:='SW_', sDescr:='Sollwert');
  LblFunctions_SetpointComfortHeating                            :FB_BA_Label:=( sObjName:='SW_', sDescr:='Sollwert Comfort Heizen');
  LblFunctions_SetpointPreComfortHeating                         :FB_BA_Label:=( sObjName:='SW_', sDescr:='Sollwert Pre-comfort Heizen');
  LblFunctions_SetpointEconomyHeating                            :FB_BA_Label:=( sObjName:='SW_', sDescr:='Sollwert Economy Heizen');
  LblFunctions_SetpointProtectionHeating                         :FB_BA_Label:=( sObjName:='SW_', sDescr:='Sollwert Protection Heizen');
  LblFunctions_SetpointComfortCooling                            :FB_BA_Label:=( sObjName:='SW_', sDescr:='Sollwert Comfort Kühlen');
  LblFunctions_SetpointPreComfortCooling                         :FB_BA_Label:=( sObjName:='SW_', sDescr:='Sollwert Pre-comfort Kühlen');
  LblFunctions_SetpointEconomyCooling                            :FB_BA_Label:=( sObjName:='SW_', sDescr:='Sollwert Economy Kühlen');
  LblFunctions_SetpointProtectionCooling                         :FB_BA_Label:=( sObjName:='SW_', sDescr:='Sollwert Protection Kühlen');
  LblFunctions_SetpointBase                                      :FB_BA_Label:=( sObjName:='SWB', sDescr:='Basissollwert');
  LblFunctions_SetpointHeating                                   :FB_BA_Label:=( sObjName:='SWH', sDescr:='Sollwert Heizen');
  LblFunctions_SetpointCooling                                   :FB_BA_Label:=( sObjName:='SWK', sDescr:='Sollwert Kühlen');
  LblFunctions_SetpointMaximum                                   :FB_BA_Label:=( sObjName:='SWX', sDescr:='Sollwert, maximal');
  LblFunctions_SetpointMechanical                                :FB_BA_Label:=( sObjName:='SWM', sDescr:='Sollwert, mechanisch');
  LblFunctions_SetpointMinimum                                   :FB_BA_Label:=( sObjName:='SWI', sDescr:='Sollwert, minimal');
  LblFunctions_SetpointNight                                     :FB_BA_Label:=( sObjName:='SWN', sDescr:='Sollwert Nacht');
  LblFunctions_SetpointDay                                       :FB_BA_Label:=( sObjName:='SWT', sDescr:='Sollwert Tag');
  LblFunctions_SetpointAdjuster                                  :FB_BA_Label:=( sObjName:='SWV', sDescr:='Sollwertversteller');
  LblFunctions_SetpointAdjustmentMechanical                      :FB_BA_Label:=( sObjName:='SVM', sDescr:='Sollwertverstellung, mechanisch');
  LblFunctions_Selection                                         :FB_BA_Label:=( sObjName:='AUS', sDescr:='Auswahl');
  LblFunctions_Status                                            :FB_BA_Label:=( sObjName:='STA', sDescr:='Status');
  LblFunctions_ControlSignal                                     :FB_BA_Label:=( sObjName:='ST_', sDescr:='Stellsignal');
  LblFunctions_Fault                                             :FB_BA_Label:=( sObjName:='SM_', sDescr:='Störung');
  LblFunctions_FaultFuse                                         :FB_BA_Label:=( sObjName:='SM_', sDescr:='Sicherung Störung ');
  LblFunctions_Button                                            :FB_BA_Label:=( sObjName:='TS_', sDescr:='Taster');
  LblFunctions_DeadZone                                          :FB_BA_Label:=( sObjName:='TZ_', sDescr:='Totzone');
  LblFunctions_ObjectTrendLogMultiple                            :FB_BA_Label:=( sObjName:='TRM', sDescr:='Trend-Log-Multiple-Objekt');
  LblFunctions_ObjectTrendLog                                    :FB_BA_Label:=( sObjName:='TR_', sDescr:='Trend-Log-Objekt');
  LblFunctions_AmplificationController                           :FB_BA_Label:=( sObjName:='KP_', sDescr:='Verstärkung Regler');
  LblFunctions_RetentionPeriod                                   :FB_BA_Label:=( sObjName:='TV_', sDescr:='Vorhaltezeit');
  LblFunctions_MaintenanceMessage                                :FB_BA_Label:=( sObjName:='WM_', sDescr:='Wartungsmeldung');
  LblFunctions_Efficiency                                        :FB_BA_Label:=( sObjName:='WG_', sDescr:='Wirkungsgrad');
  LblFunctions_CountValue                                        :FB_BA_Label:=( sObjName:='ZW_', sDescr:='Zählwert');
  LblFunctions_TimeProgram                                       :FB_BA_Label:=( sObjName:='ZPR', sDescr:='Zeitprogramm');
// Beckhoff Skalierung
  LblFunctions_ValueX1                                           :FB_BA_Label:=( sObjName:='SPX', sDescr:='Wert Stützpunkt [X1]');
  LblFunctions_ValueX2                                           :FB_BA_Label:=( sObjName:='SPX', sDescr:='Wert Stützpunkt [X2]');
  LblFunctions_ValueX3                                           :FB_BA_Label:=( sObjName:='SPX', sDescr:='Wert Stützpunkt [X3]');
  LblFunctions_ValueX4                                           :FB_BA_Label:=( sObjName:='SPX', sDescr:='Wert Stützpunkt [X4]');
  LblFunctions_ValueX5                                           :FB_BA_Label:=( sObjName:='SPX', sDescr:='Wert Stützpunkt [X5]');
  LblFunctions_ValueX6                                           :FB_BA_Label:=( sObjName:='SPX', sDescr:='Wert Stützpunkt [X6]');
  LblFunctions_ValueX7                                           :FB_BA_Label:=( sObjName:='SPX', sDescr:='Wert Stützpunkt [X7]');
  LblFunctions_ValueY1                                           :FB_BA_Label:=( sObjName:='SPY', sDescr:='Wert Stützpunkt [Y1]');
  LblFunctions_ValueY2                                           :FB_BA_Label:=( sObjName:='SPY', sDescr:='Wert Stützpunkt [Y2]');
  LblFunctions_ValueY3                                           :FB_BA_Label:=( sObjName:='SPY', sDescr:='Wert Stützpunkt [Y3]');
  LblFunctions_ValueY2_3                                         :FB_BA_Label:=( sObjName:='SPY', sDescr:='Wert Stützpunkt [Y2-Y3]');
  LblFunctions_ValueY4                                           :FB_BA_Label:=( sObjName:='SPY', sDescr:='Wert Stützpunkt [Y4]');
  LblFunctions_ValueY5                                           :FB_BA_Label:=( sObjName:='SPY', sDescr:='Wert Stützpunkt [Y5]');
  LblFunctions_ValueY6                                           :FB_BA_Label:=( sObjName:='SPY', sDescr:='Wert Stützpunkt [Y6]');
  LblFunctions_ValueY7                                           :FB_BA_Label:=( sObjName:='SPY', sDescr:='Wert Stützpunkt [Y7]');
  LblFunctions_SuppyAirTempSetpointHeaterCalc                    :FB_BA_Label:=( sObjName:='SWC', sDescr:='Zulufttemperatursollwert Erhitzer errechnet');
  LblFunctions_SuppyAirTempSetpointCoolerCalc                    :FB_BA_Label:=( sObjName:='SWC', sDescr:='Zulufttemperatursollwert Kühler errechnet');
  LblFunctions_SuppyAirTempSetpointERCCalc                       :FB_BA_Label:=( sObjName:='SWC', sDescr:='Zulufttemperatursollwert ERG errechnet');
END_VAR

// ---- Templates/GVLs/DPAD/Labels/1033/LblAggregates1033.TcGVL
{region '#Template'}
	{attribute 'Version' := '1.0.0.0'}
	{attribute 'Tags' := '"LCID": "1031", "Text": "GVL, AKS, Labels, ObjectName, Description"'}
	{attribute 'Tags' := '"LCID": "1033", "Text": "GVL, DPAD, Labels, ObjectName, Description"'}
	{attribute 'Description' := '"LCID": "1031", "Text": "Anlagenkennzeichnungssystem, Labels Aggregate"'}
	{attribute 'Description' := '"LCID": "1033", "Text": "Data Point Addressing Description, Labels aggregate"'}
{endregion}
	 
